FUNCTION_BLOCK FB_LA
VAR_INPUT

	Modbus_LA		: BOOL;
END_VAR
VAR_IN_OUT
END_VAR
VAR_OUTPUT
END_VAR
VAR
(*Diagnose-Funktion stellt eine Reihe von Tests für die Überprüfung des Übertragungssystems zwischen dem Master und dem Slave,
oder für die Überprüfung der verschiedenen internen Fehlerzustände innerhalb des Slaves, zur Verfügung.*)
	LA_955_Diagnose	: FB_MBDiagnose;
	IPAddr	 		: STRING(15);(* IPv4 address of the target device *)
	TCPPort			: UINT:= MODBUS_TCP_PORT;(* Port number of the target device *)
	UnitID			: BYTE:=16#FF;(* Identification number of a serial sub-network device *)
	WriteData		: WORD;
	Execute			: BOOL;(* Rising edge at this input starts command execution *)
	Timeout			: TIME;
	SubFnc			: WORD;
	Diagnose		: BOOL;
	Diagnose_busy	: BOOL;
	Diagnose_Error	: BOOL;
	Diagnose_ErrorID: UDINT;
	Read_Data		: WORD;

(* FB_MBReadRegs*)
	(* Read 1..128 input registers (word access) *)
	LA_955_ReadRegs		: FB_MBReadRegs;
	DestAddrRR			: PVOID;(* Pointer to destination buffer *)
	LA955_RR_arrData	: ARRAY [1..26] OF INT;
	ReadRegsBusy_Modus	: BOOL;
	ReadRegsError_Modus	: BOOL;
	ReadRegsErrID_Modus	: UDINT;
	ReadRegsCount_Modus	: UDINT;

(* FB_MBReadInputs *)
	LA_955_ReadInputs		: FB_MBReadInputs;
	ReadInputsBusy_Modus	: BOOL;
	ReadInputs_Error_Modus	: BOOL;
	ReadInputsErrID_Modus	: UDINT;
	ReadInputsCount_Modus	: UDINT;
	LA955_RI_arrData		: ARRAY [1..31] OF BYTE;
	DestAddrInputs			: PVOID;(* Pointer to destination buffer *)

(* FB_MBWriteRegs *)
	LA_955_WriteRegs		: FB_MBWriteRegs;
	WriteRegsBusy_Modus		: BOOL;
	WriteRegs_Error_Modus	: BOOL;
	WriteRegsErrID_Modus	: UDINT;
    LA955_WR_arrData		: ARRAY [1..43] OF INT;
	SrcAddrWR				: PVOID;(* Pointer to source buffer *)

(* FB_MBWritecoils / Coils = einzelner Ein-/ausgang *)
	LA_955_WriteCoils		: FB_MBWriteCoils;
	WriteCoilsBusy_Modus	: BOOL;
	WriteCoils_Error_Modus	: BOOL;
	WriteCoilsErrID_Modus	: UDINT;
    LA955_WC_arrData		: ARRAY [1..42] OF BYTE;
	SrcAddrWC				: PVOID;(* Pointer to source buffer *)

	Aktivieren5			: BOOL;
	Aktivieren6			: BOOL;
	Ablufttemp			: REAL;

(* Blinker *)
	Blinker_Abfrage		: BOOL;
	T_on				: TIME:=t#2s;
	T_off				: TIME:=t#1s;
	Timer1				: TON;
	Timer2				: TON;

	{attribute 'OPC.UA.DA' := '1'}Steuerung		: ST_LA_Steuerung; 
	{attribute 'OPC.UA.DA' := '1'}Parameter		: ST_LA_Parameter; 
	{attribute 'OPC.UA.DA' := '1'}Stellwert		: ST_LA_Stellwert; 
	{attribute 'OPC.UA.DA' := '1'}Zustand			: ST_LA_Zustand;
	Zustandscheck	: FB_LA_Zustandscheck;
END_VAR
VAR // added by the converter: edge detectors and wires of the graphical bodies
    _w1, _w2, _w3, _w4, _w5, _w6, _w7, _w8, _w9, _w10, _w11, _w12, _w13, _w14, _w15, _w16, _w17, _w18, _w19, _w20, _w21, _w22, _w23, _w24, _w25, _w26, _w27, _w28, _w29, _w30, _w31, _w32 : ANY;
END_VAR

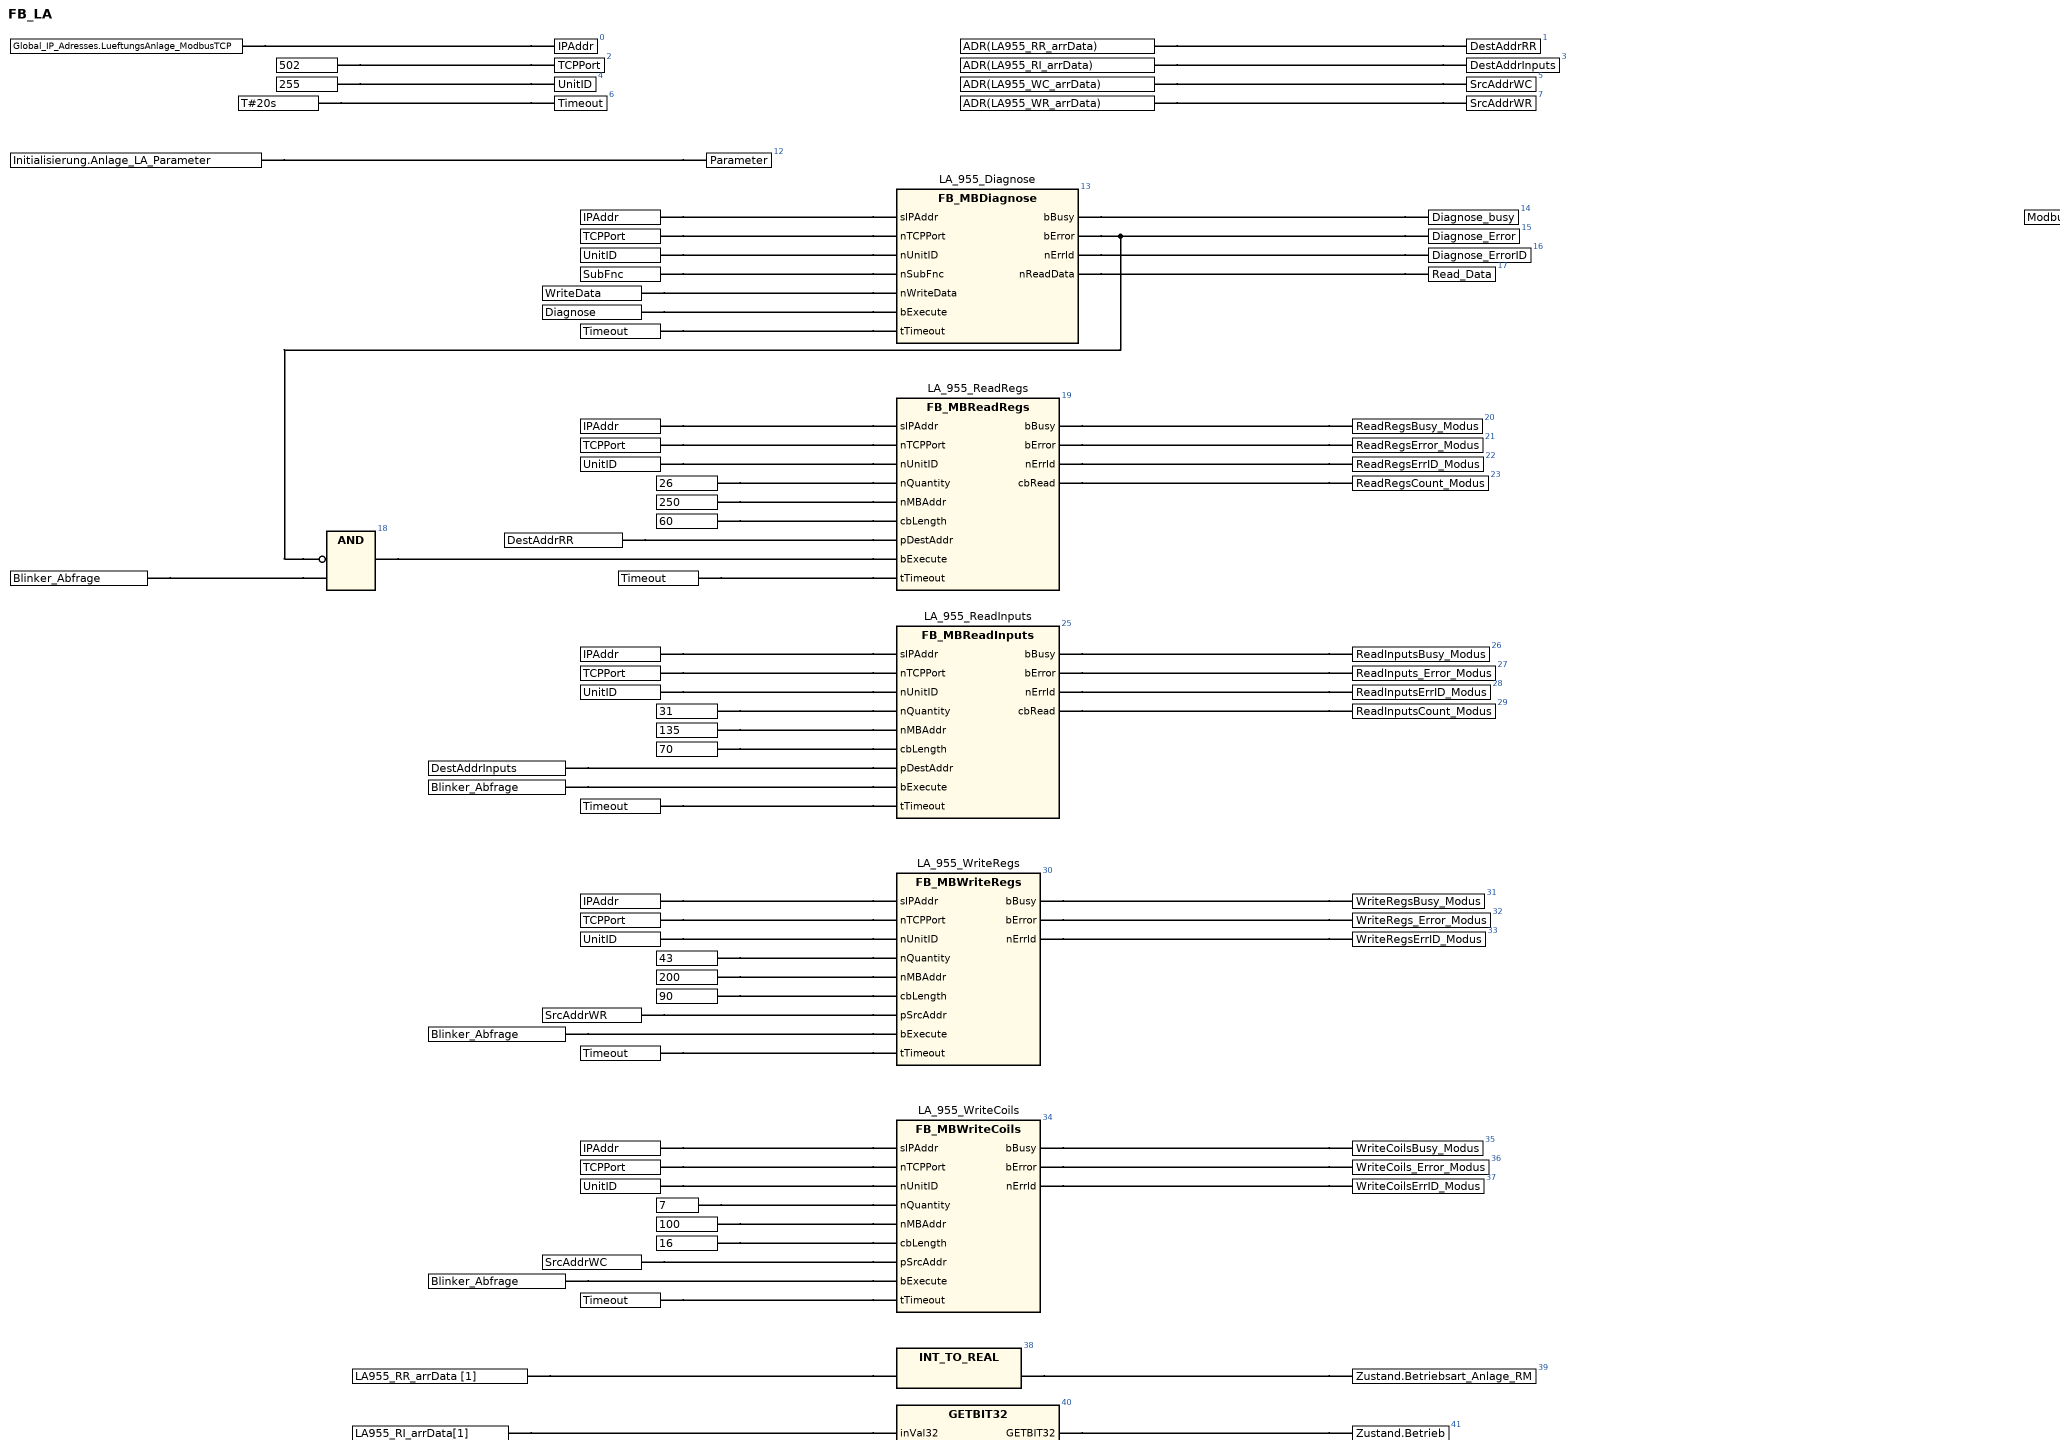
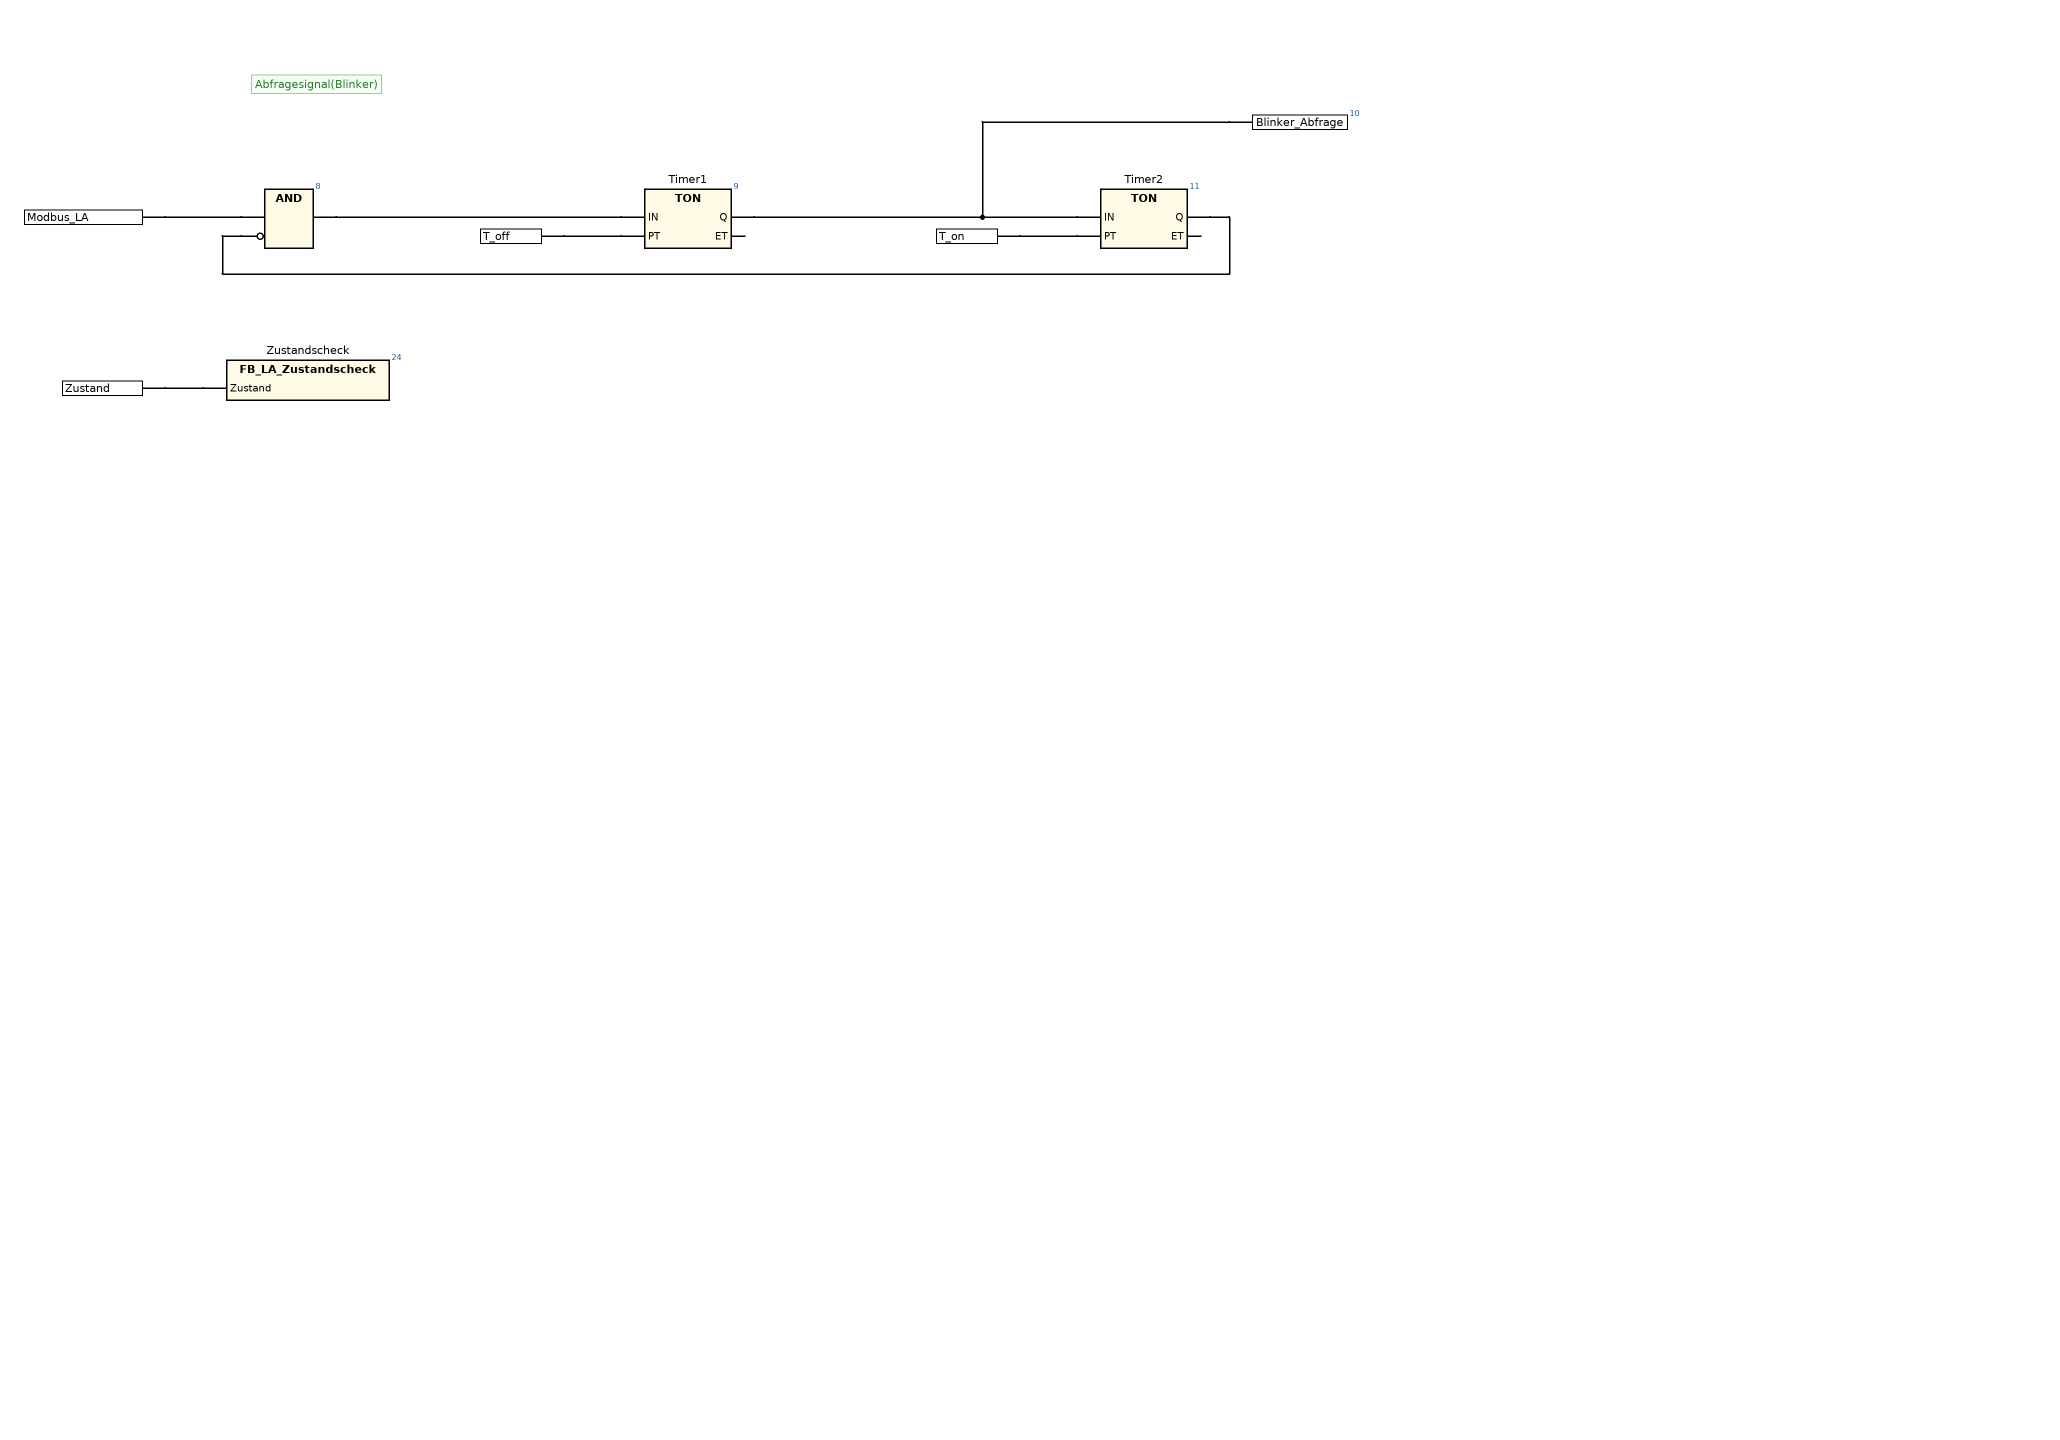
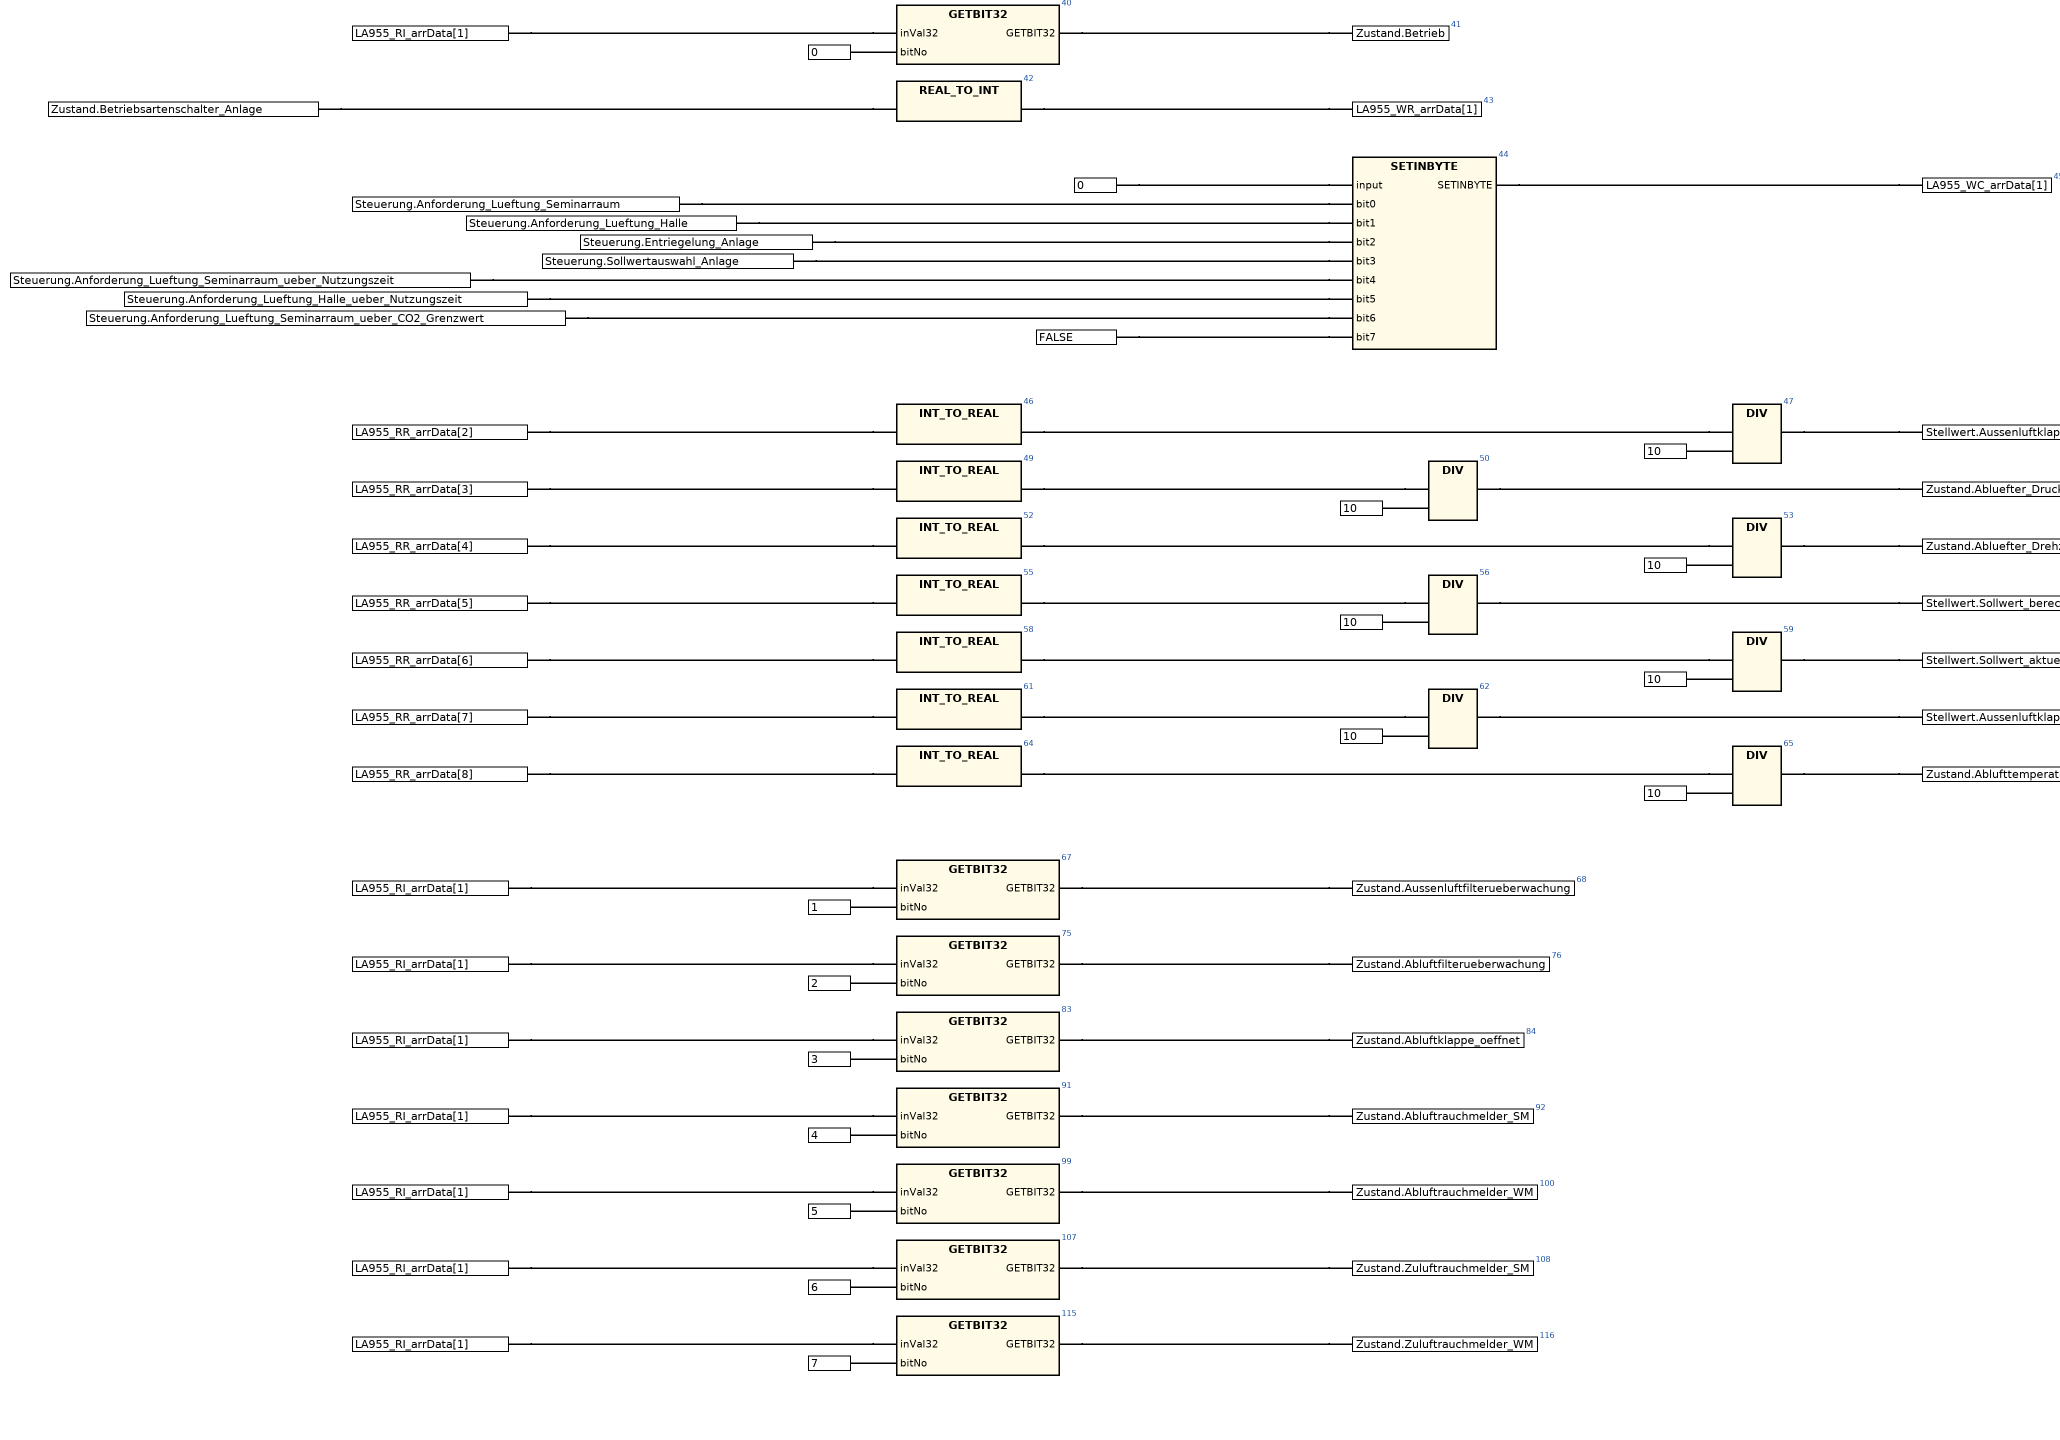
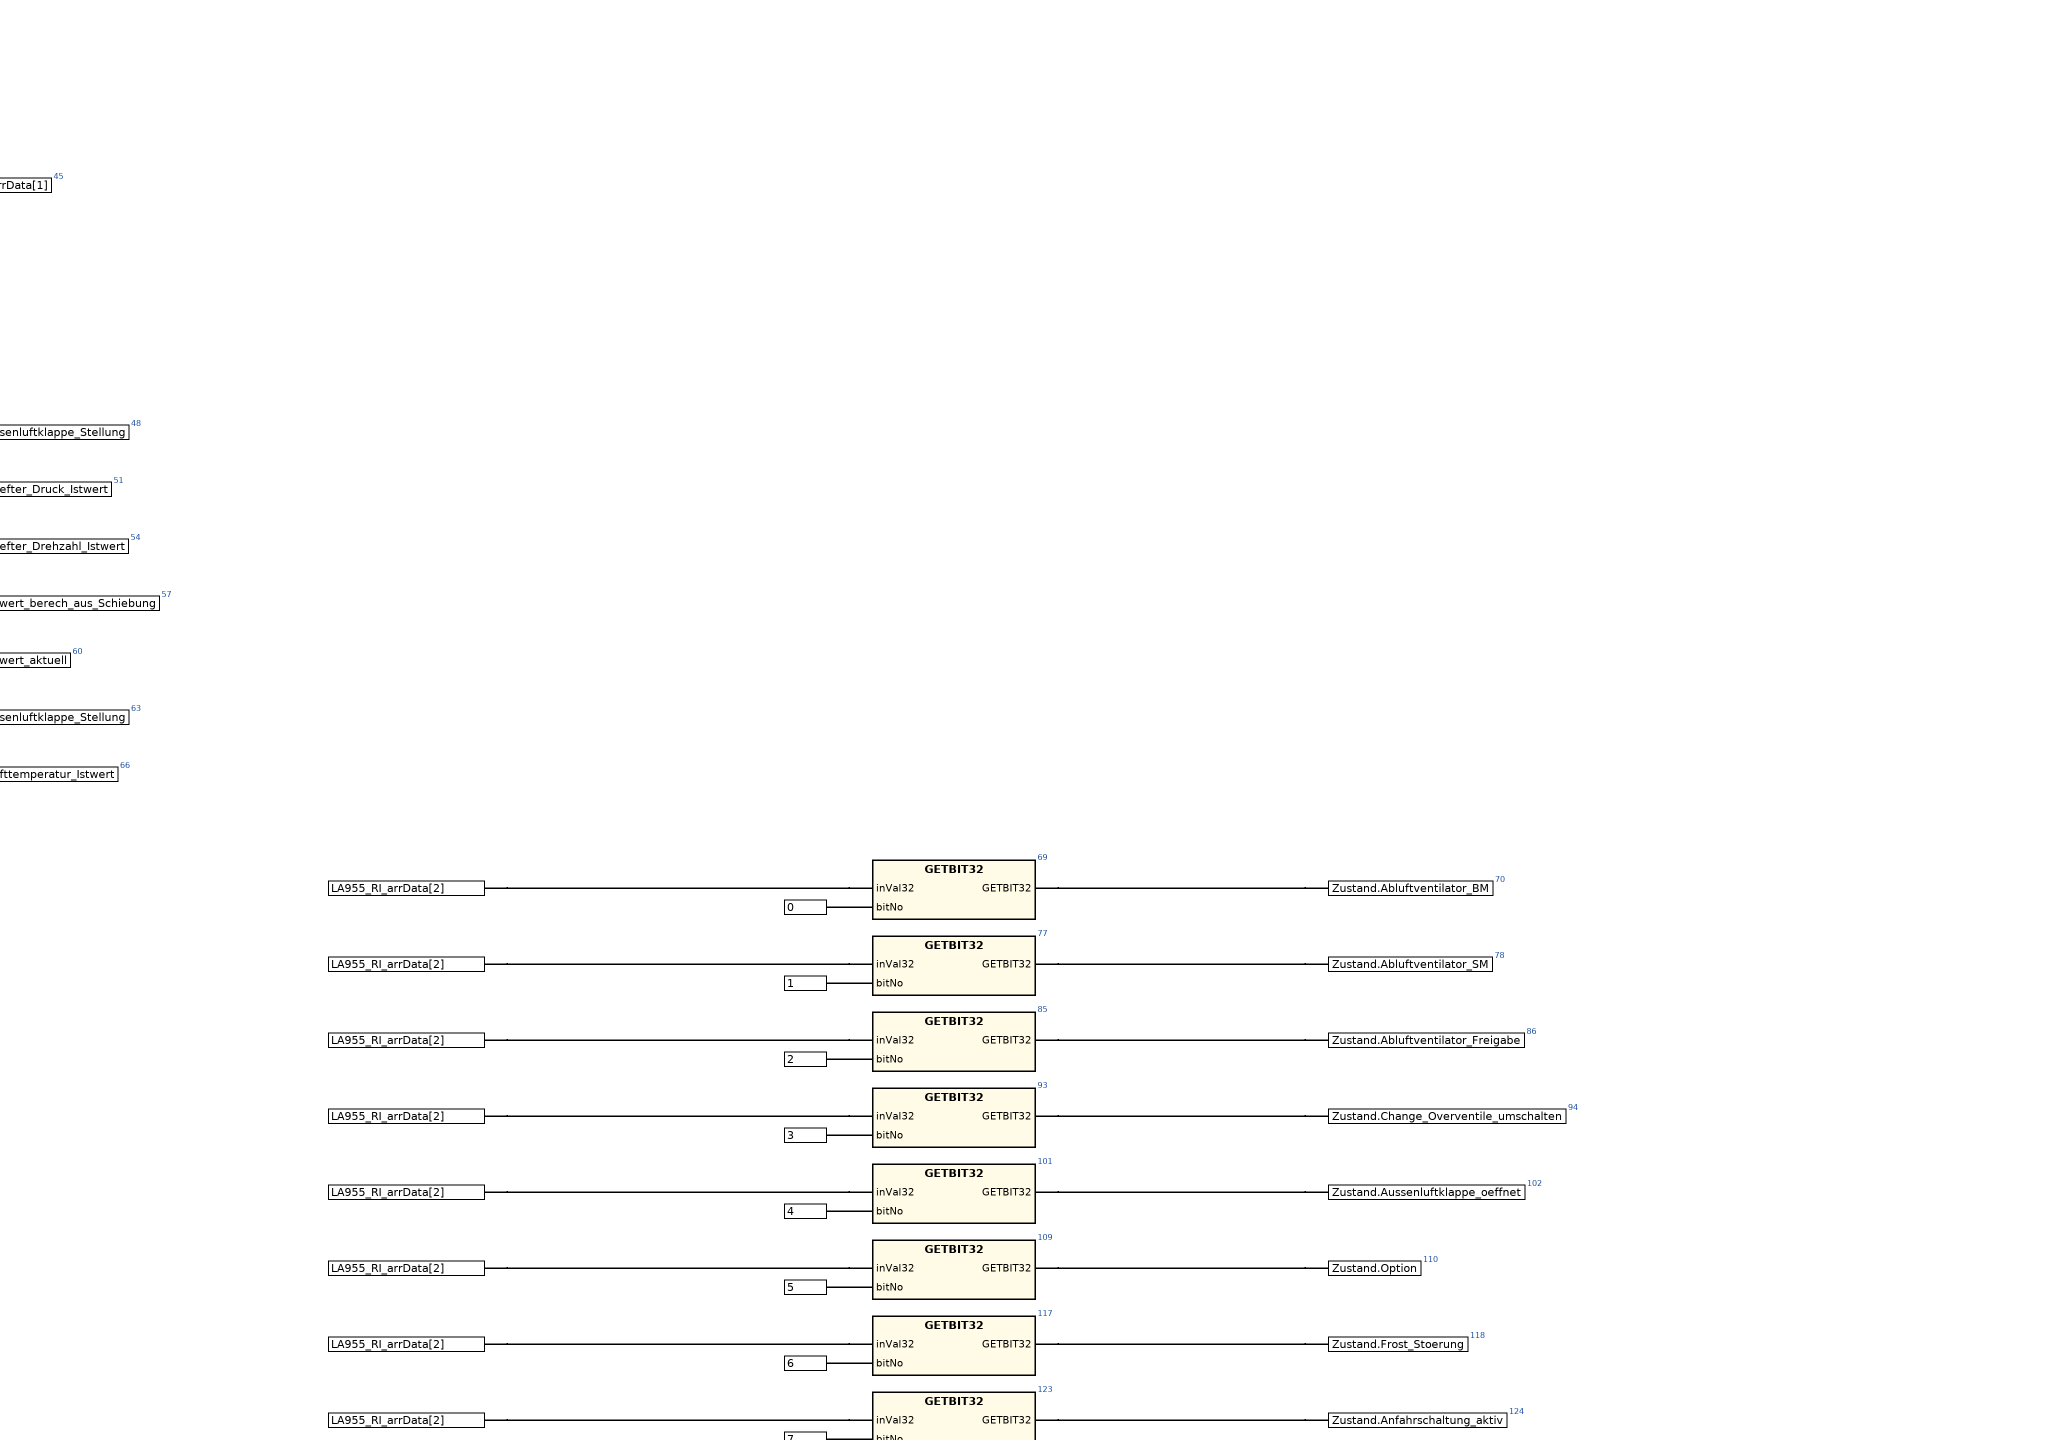
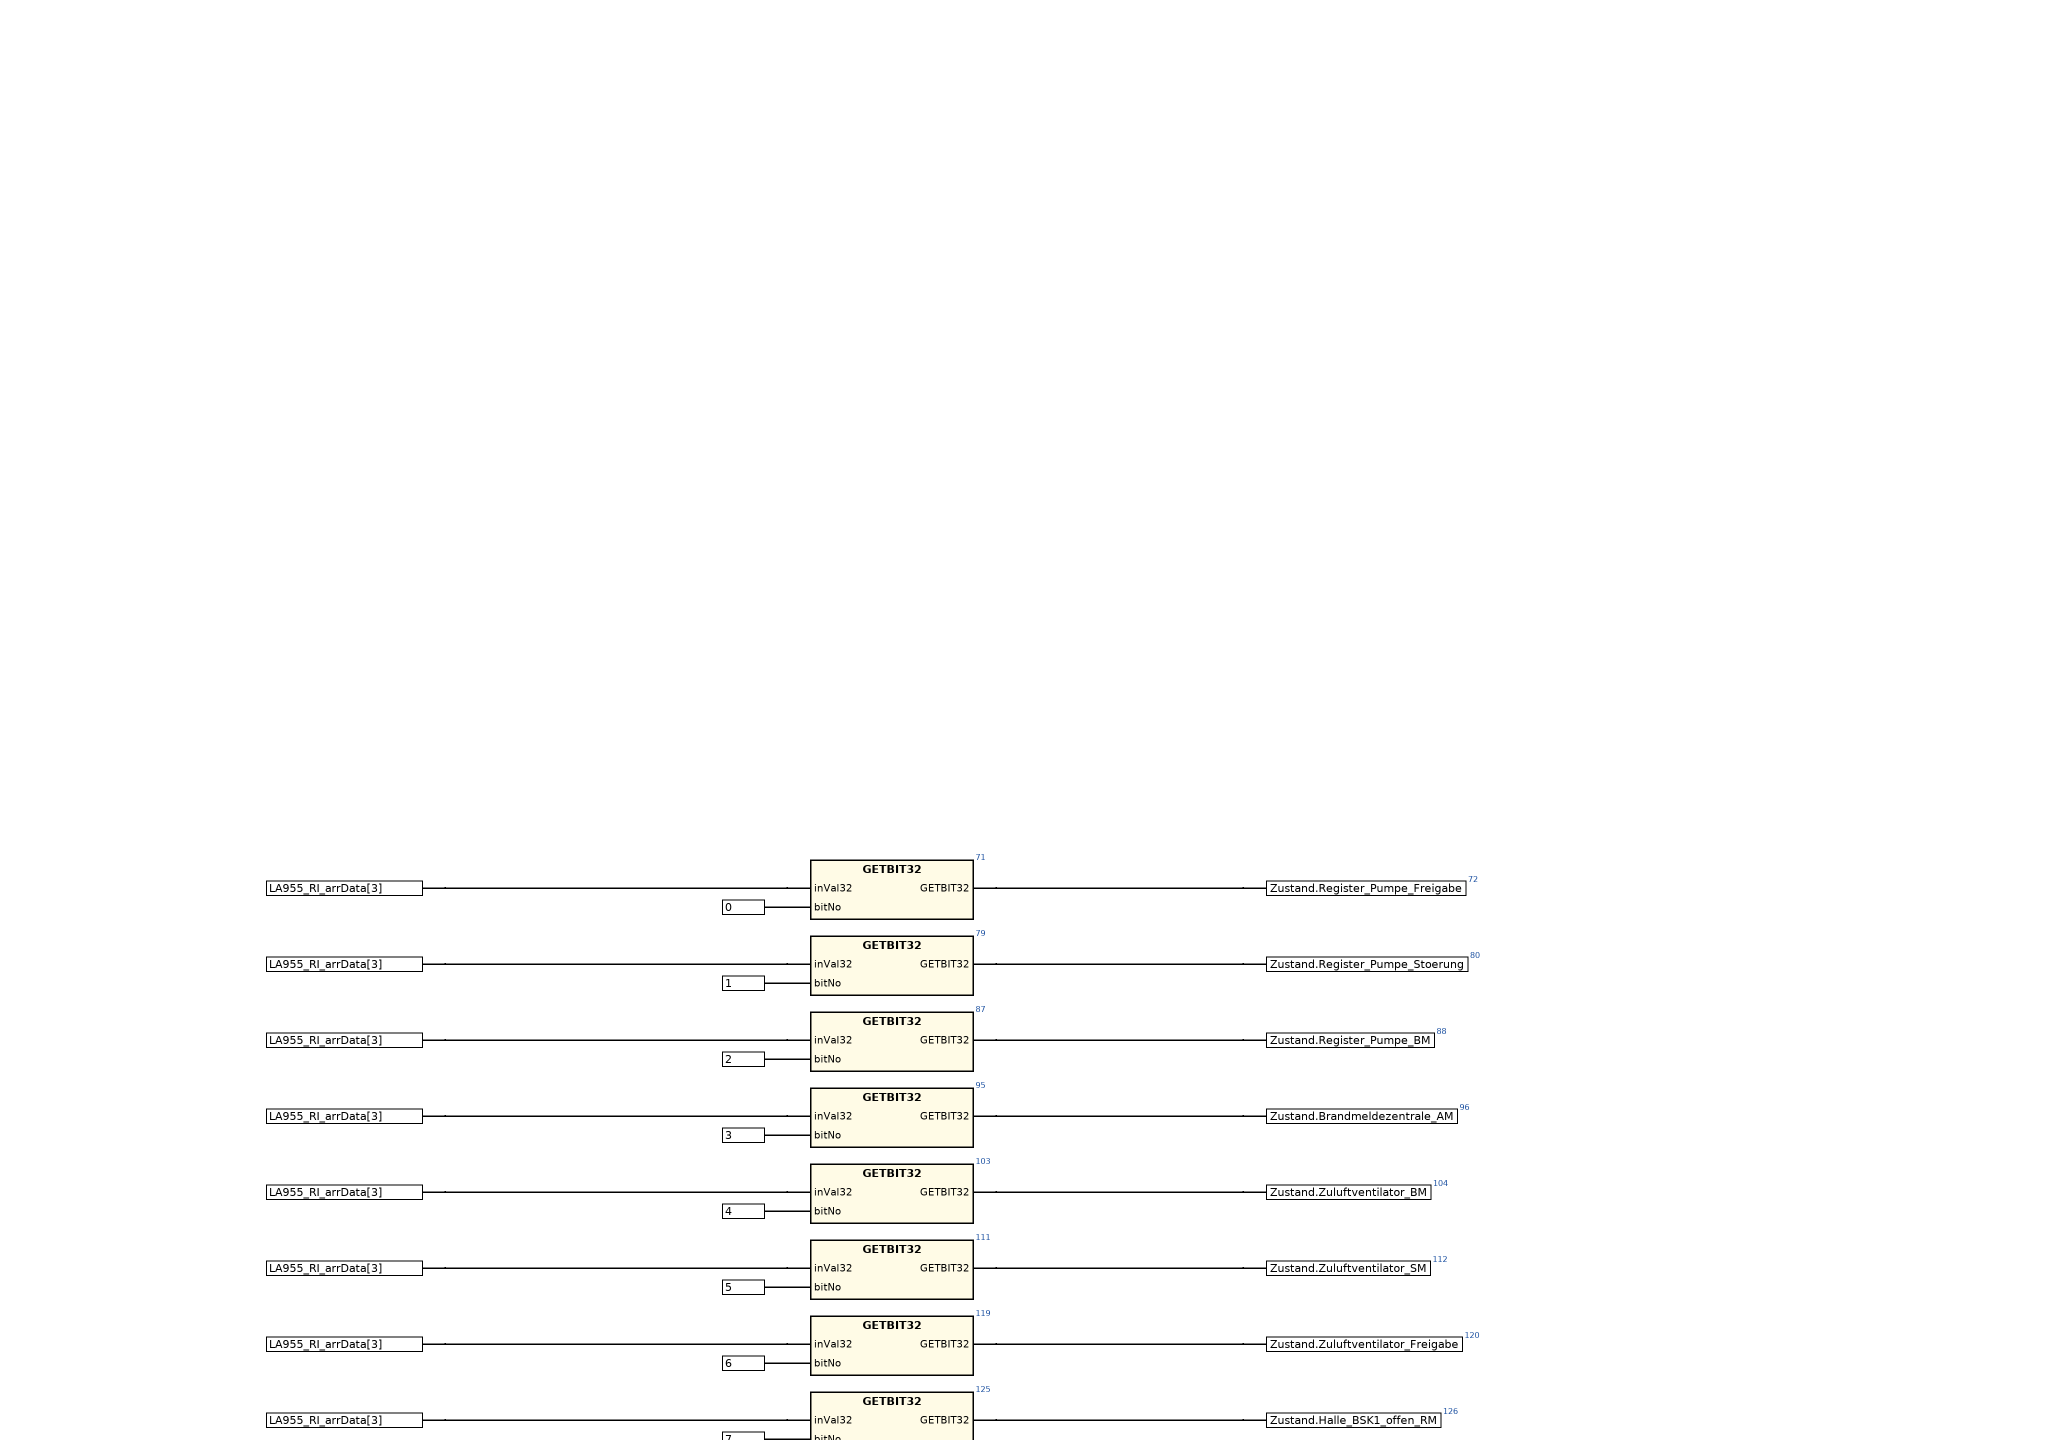
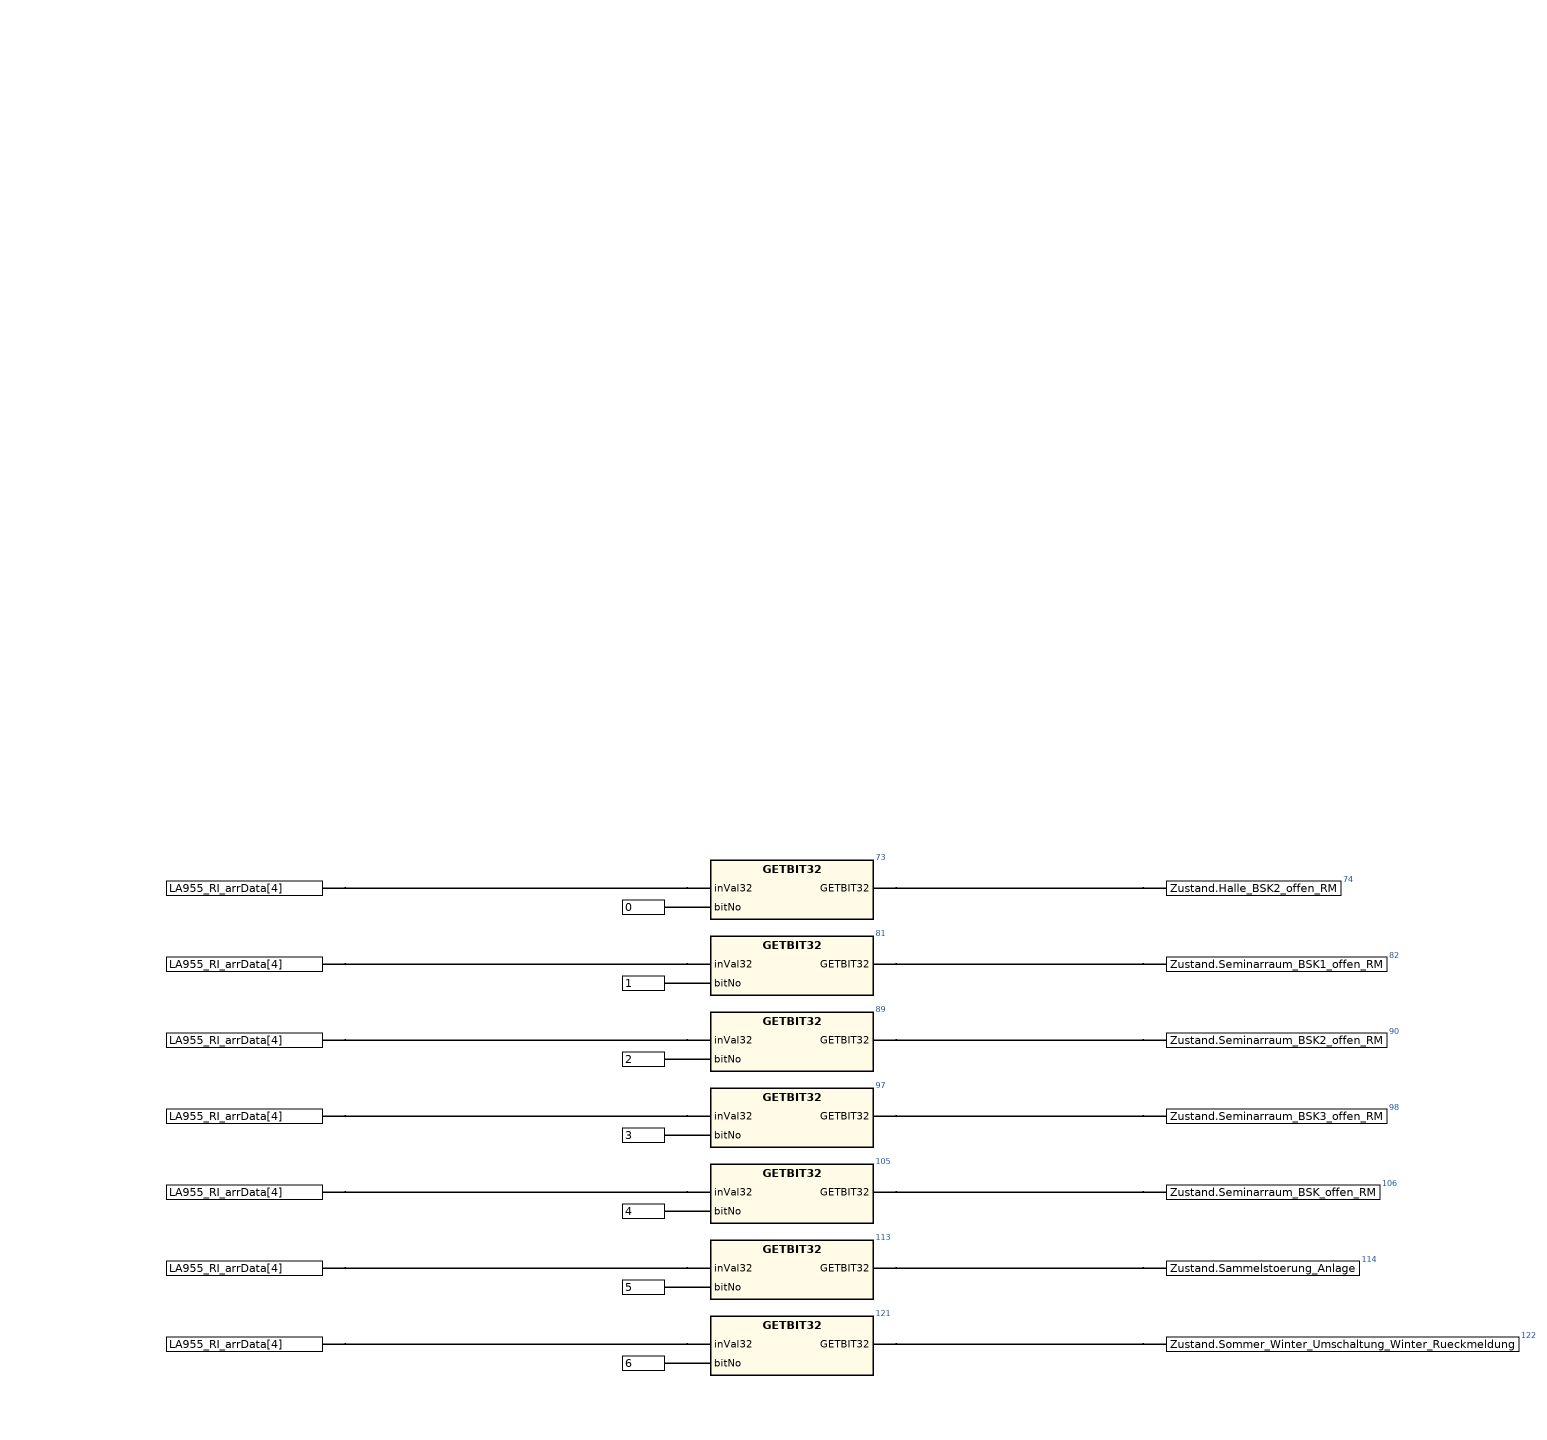
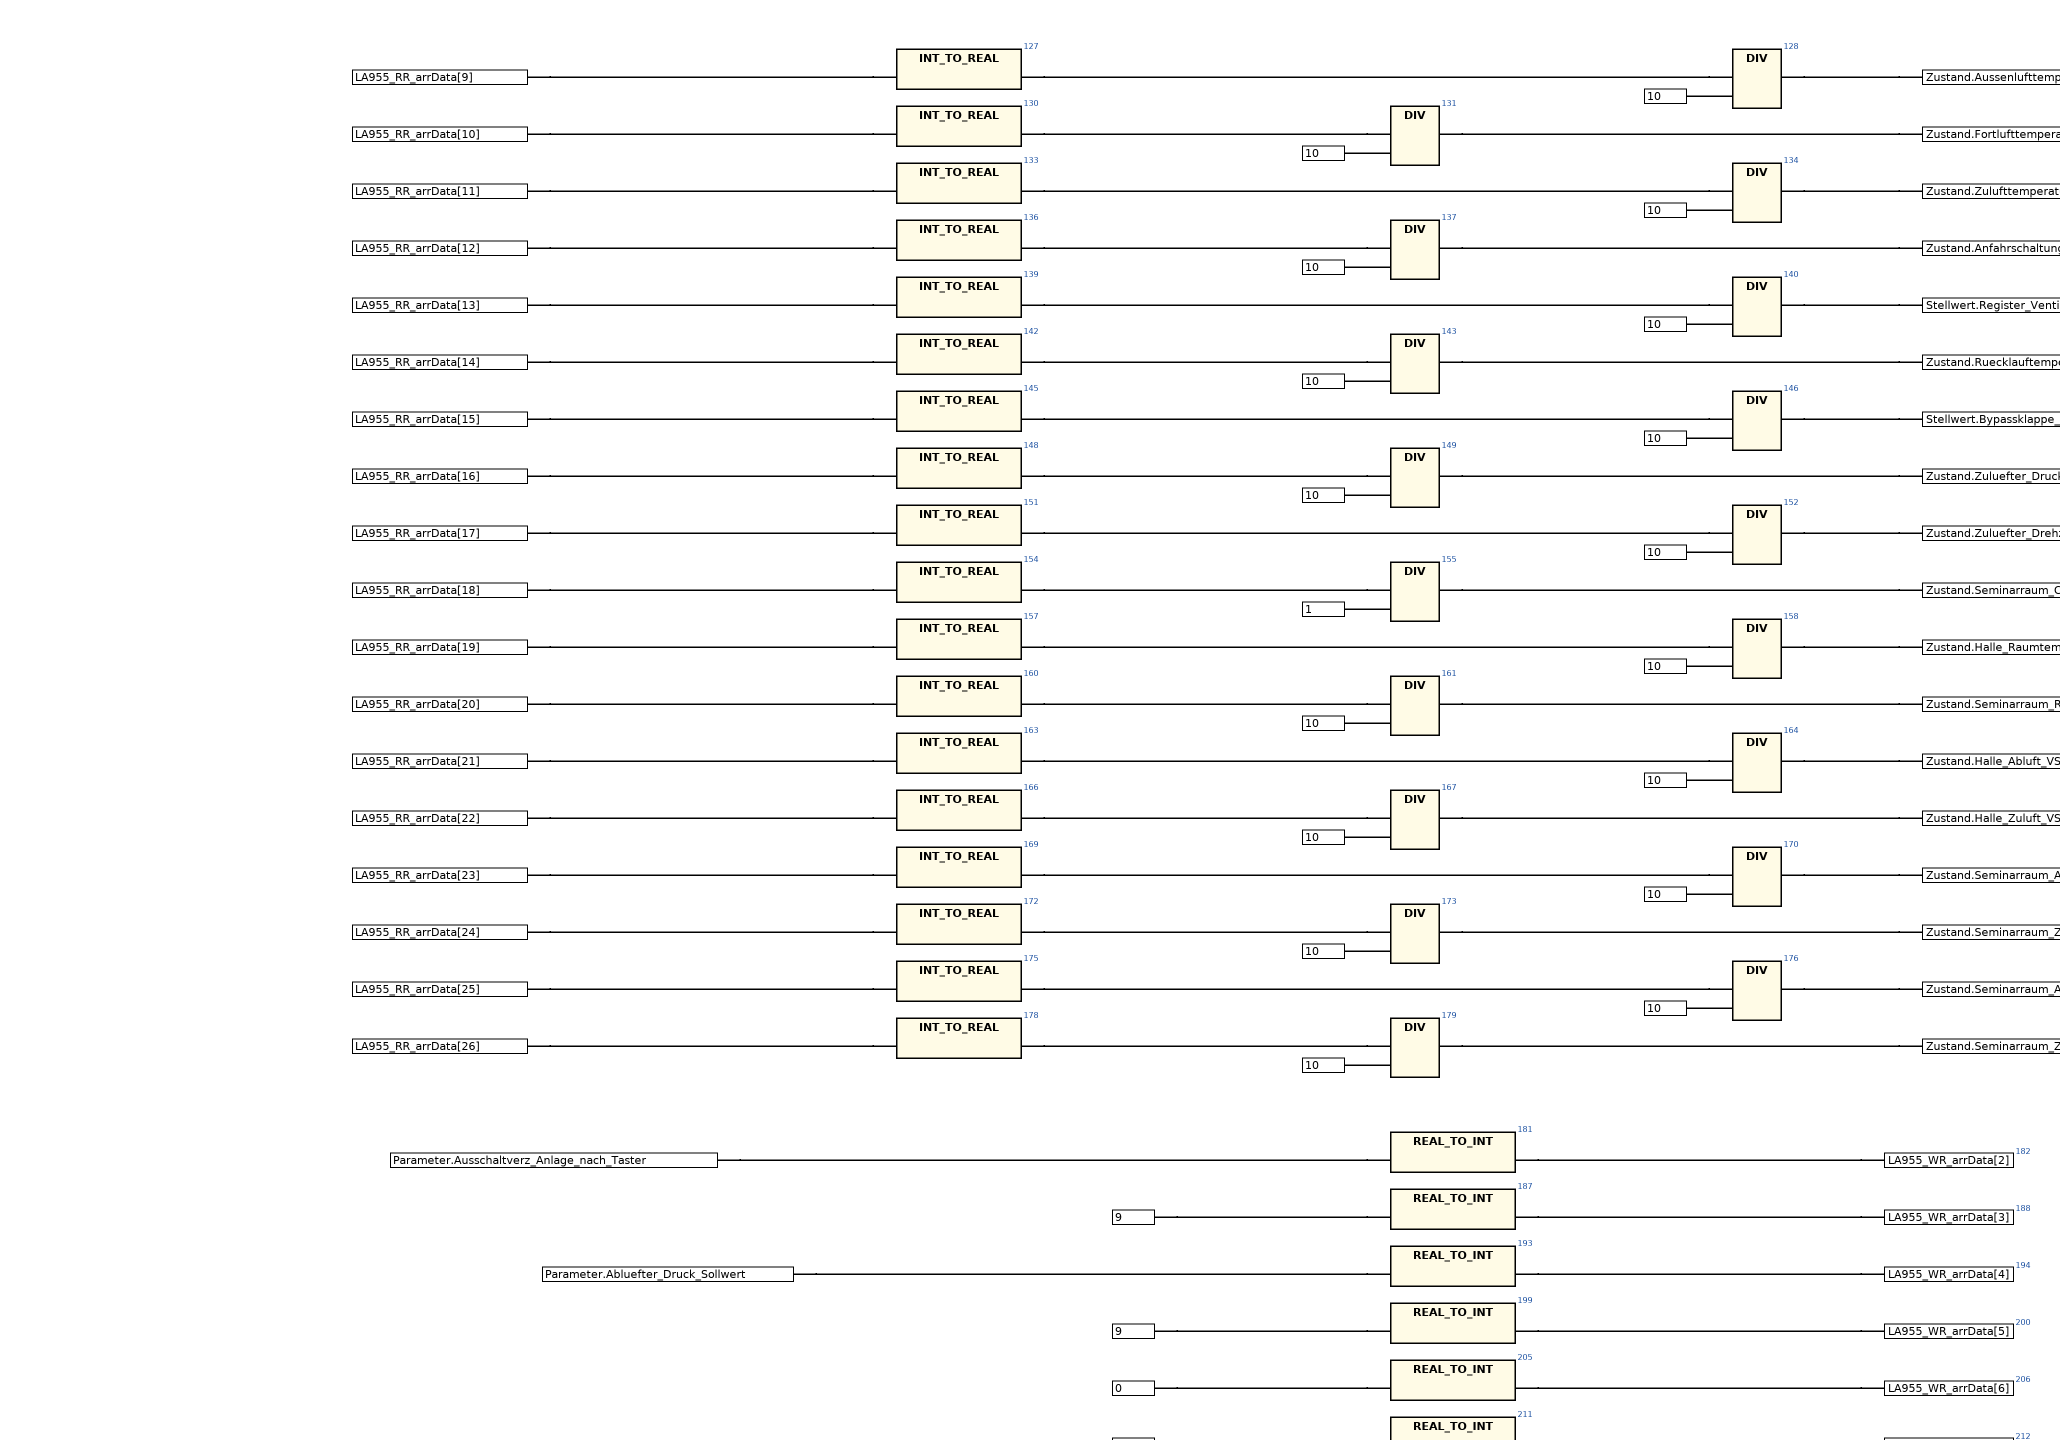
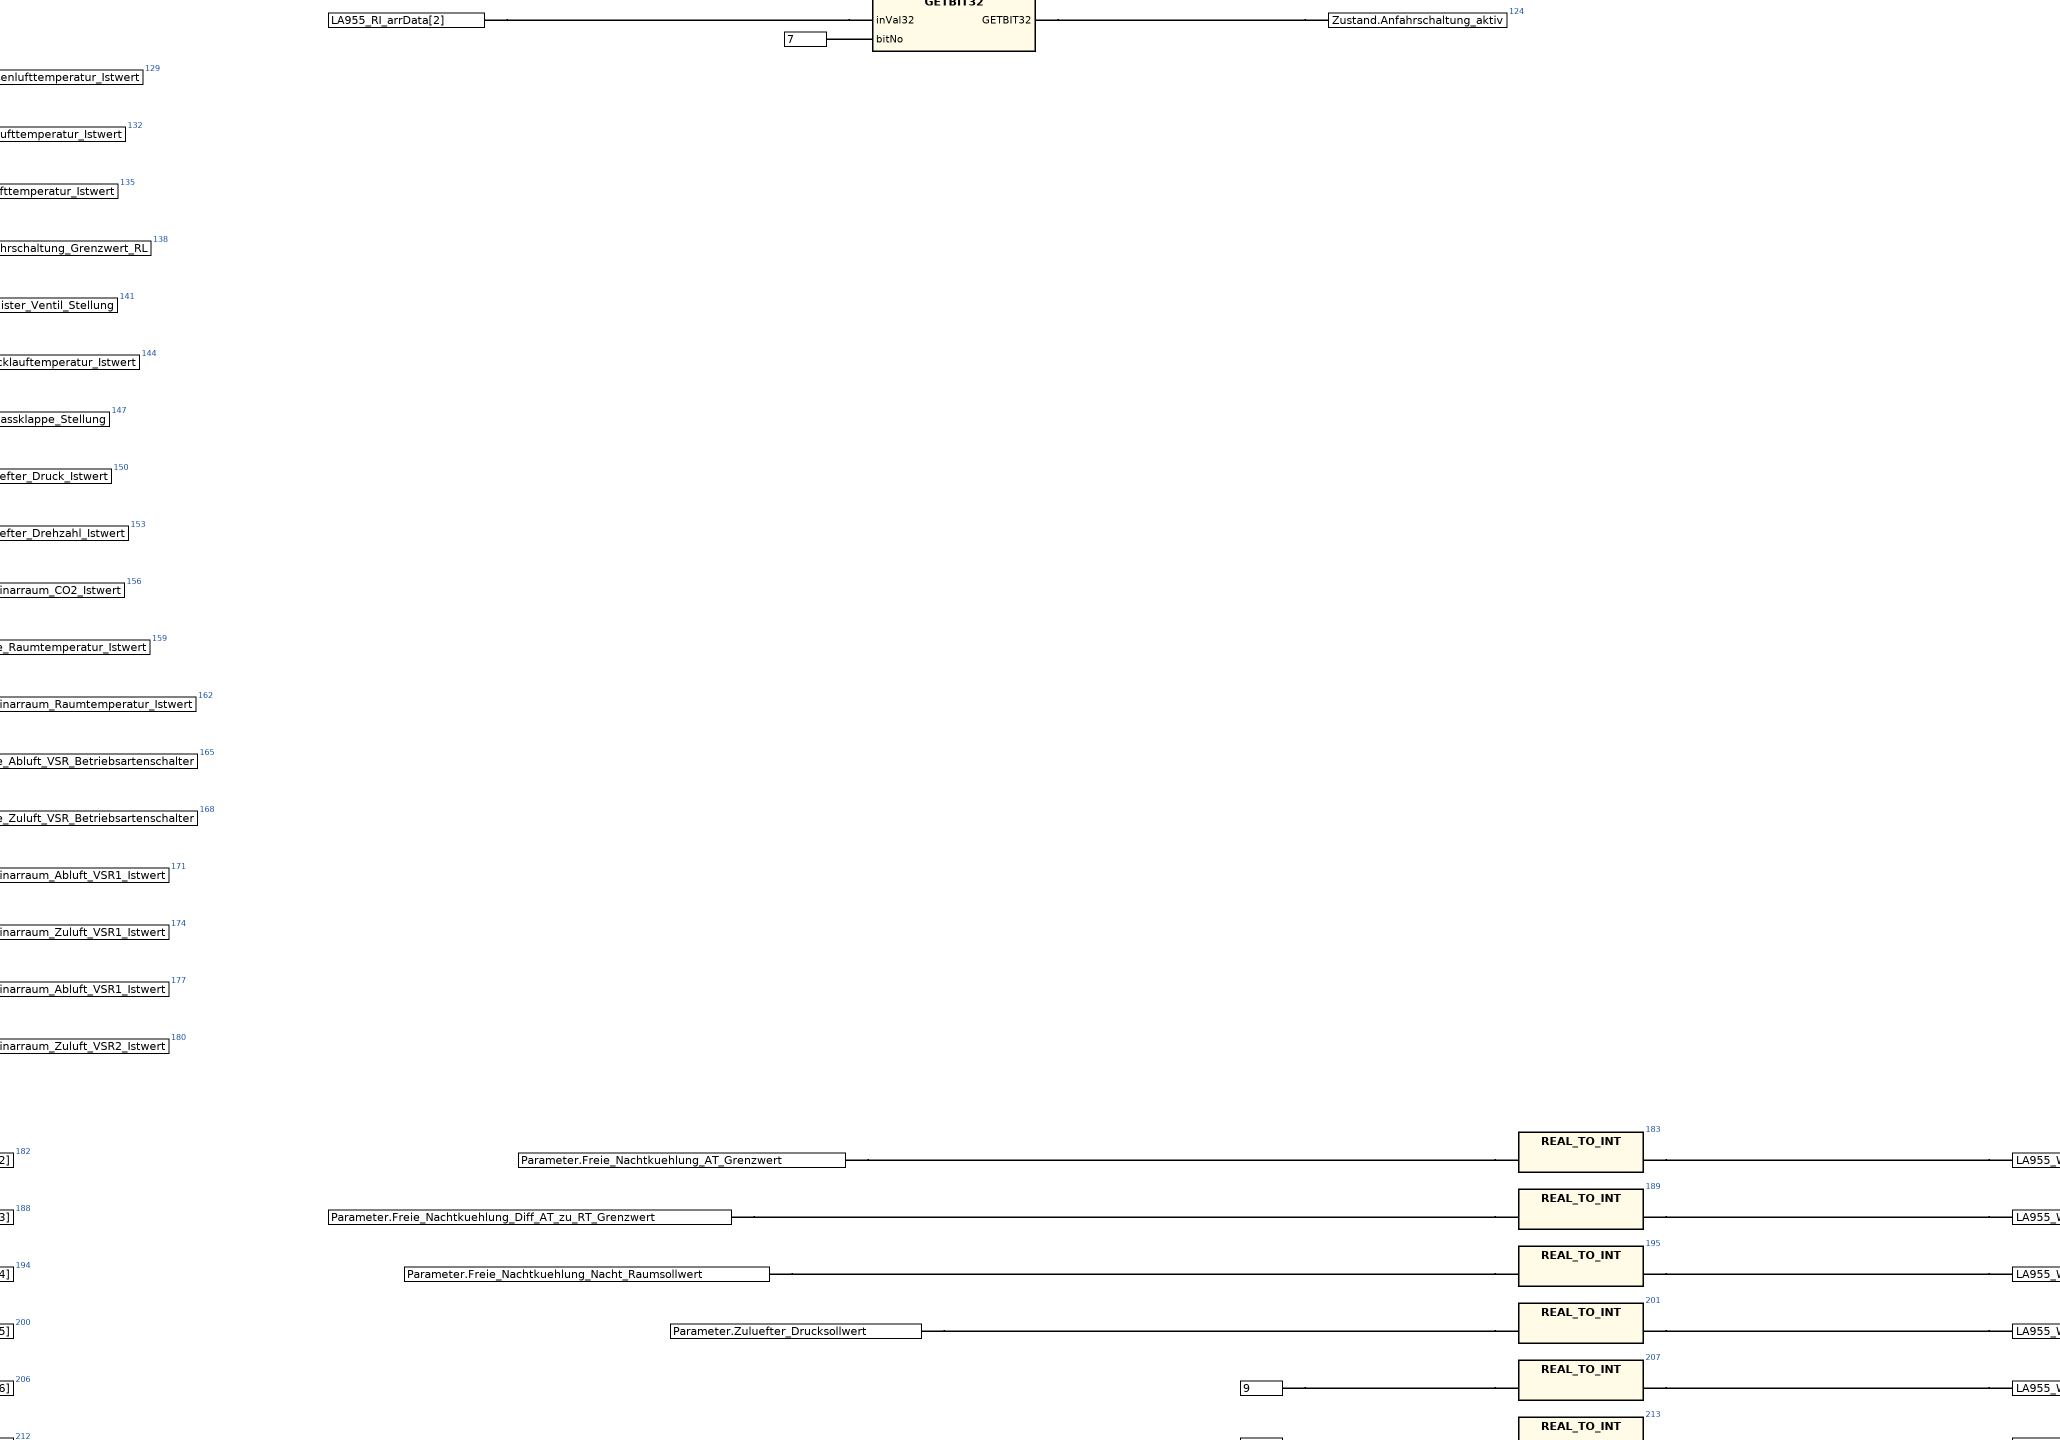
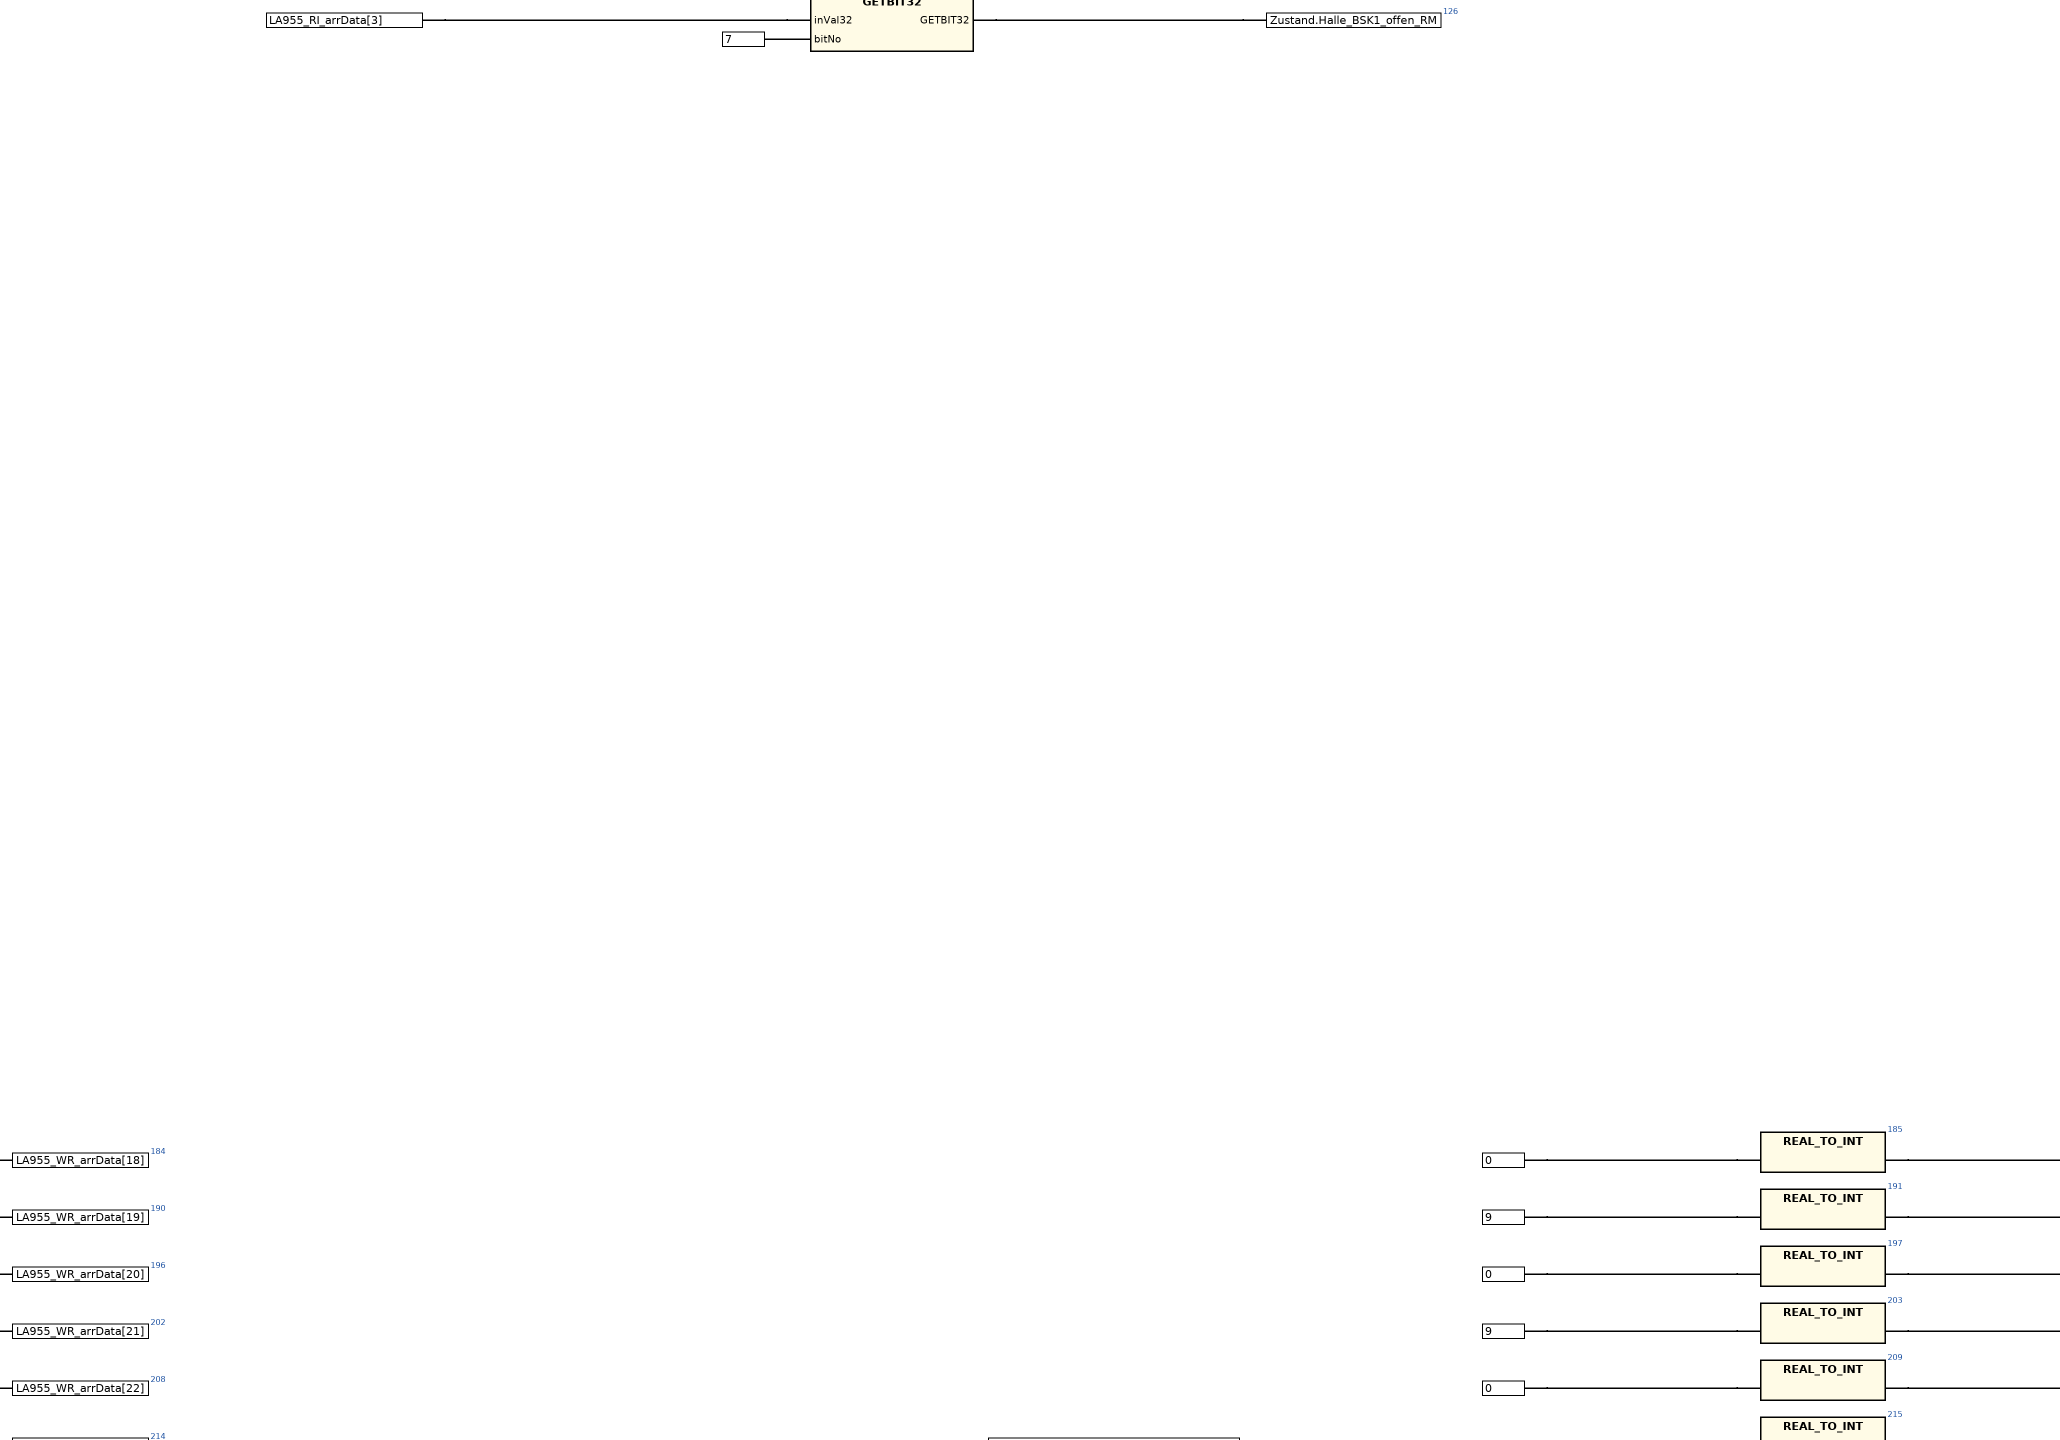
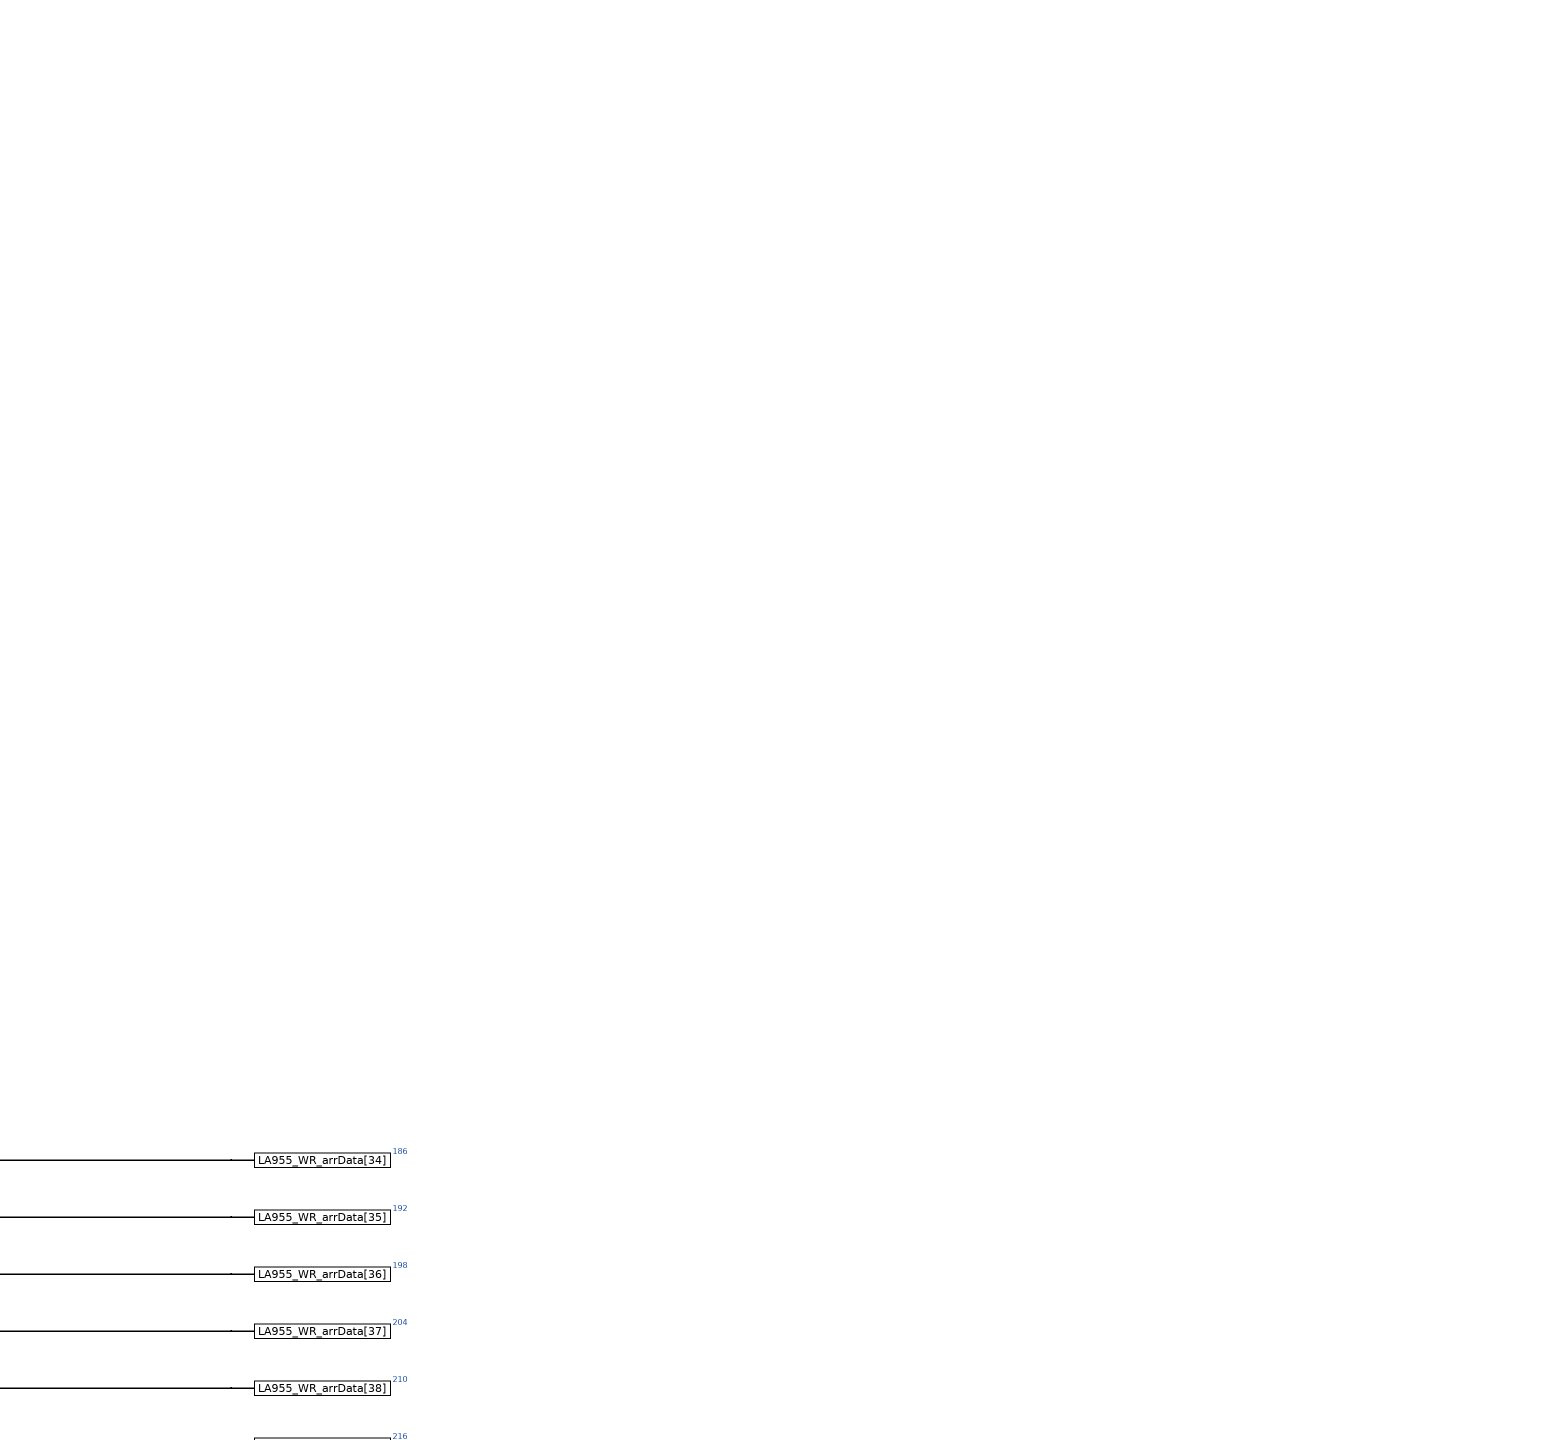
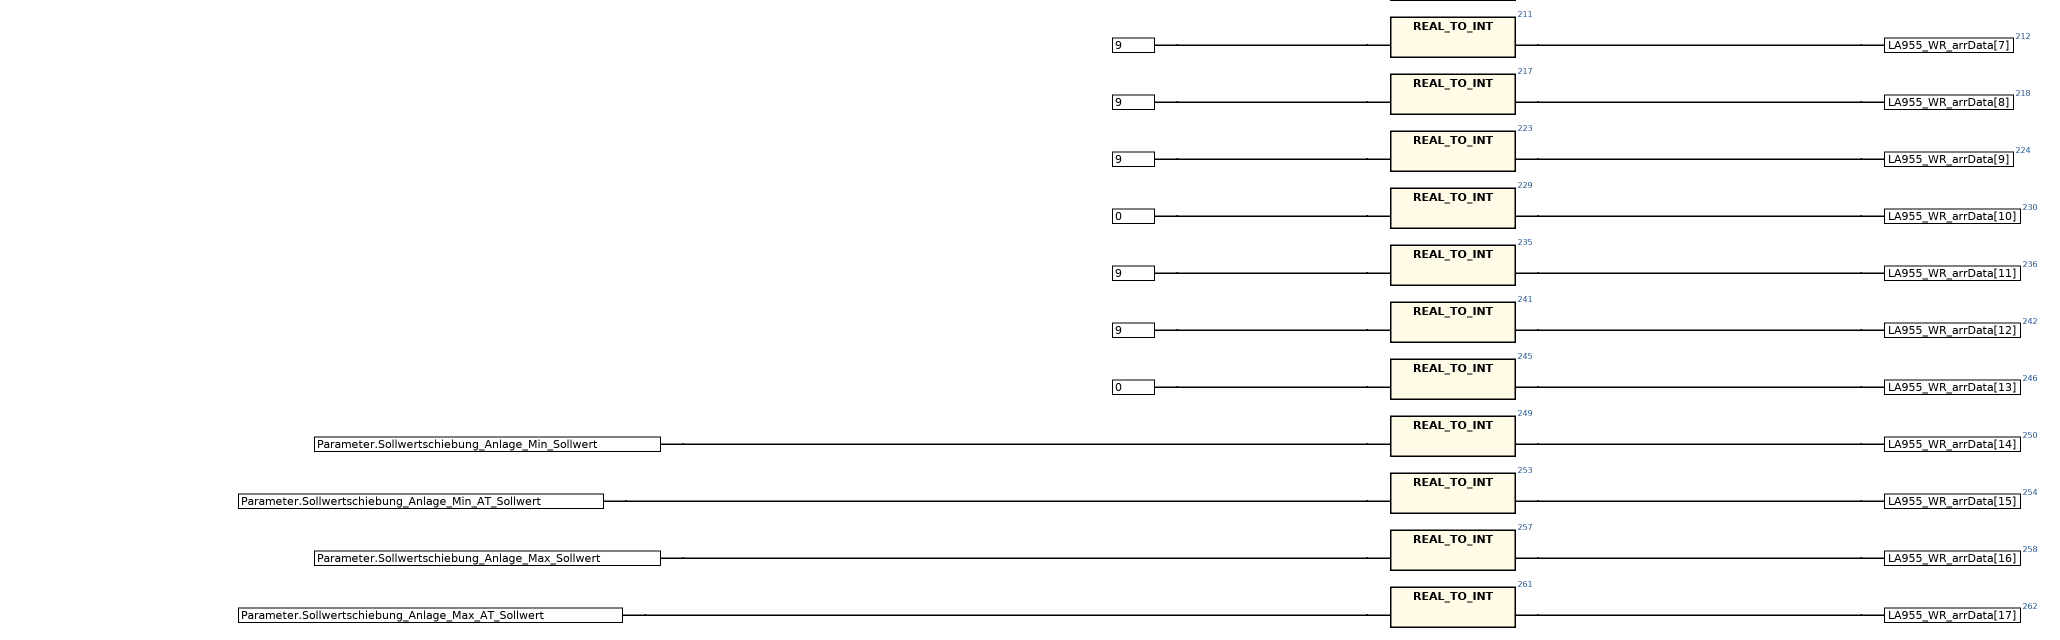
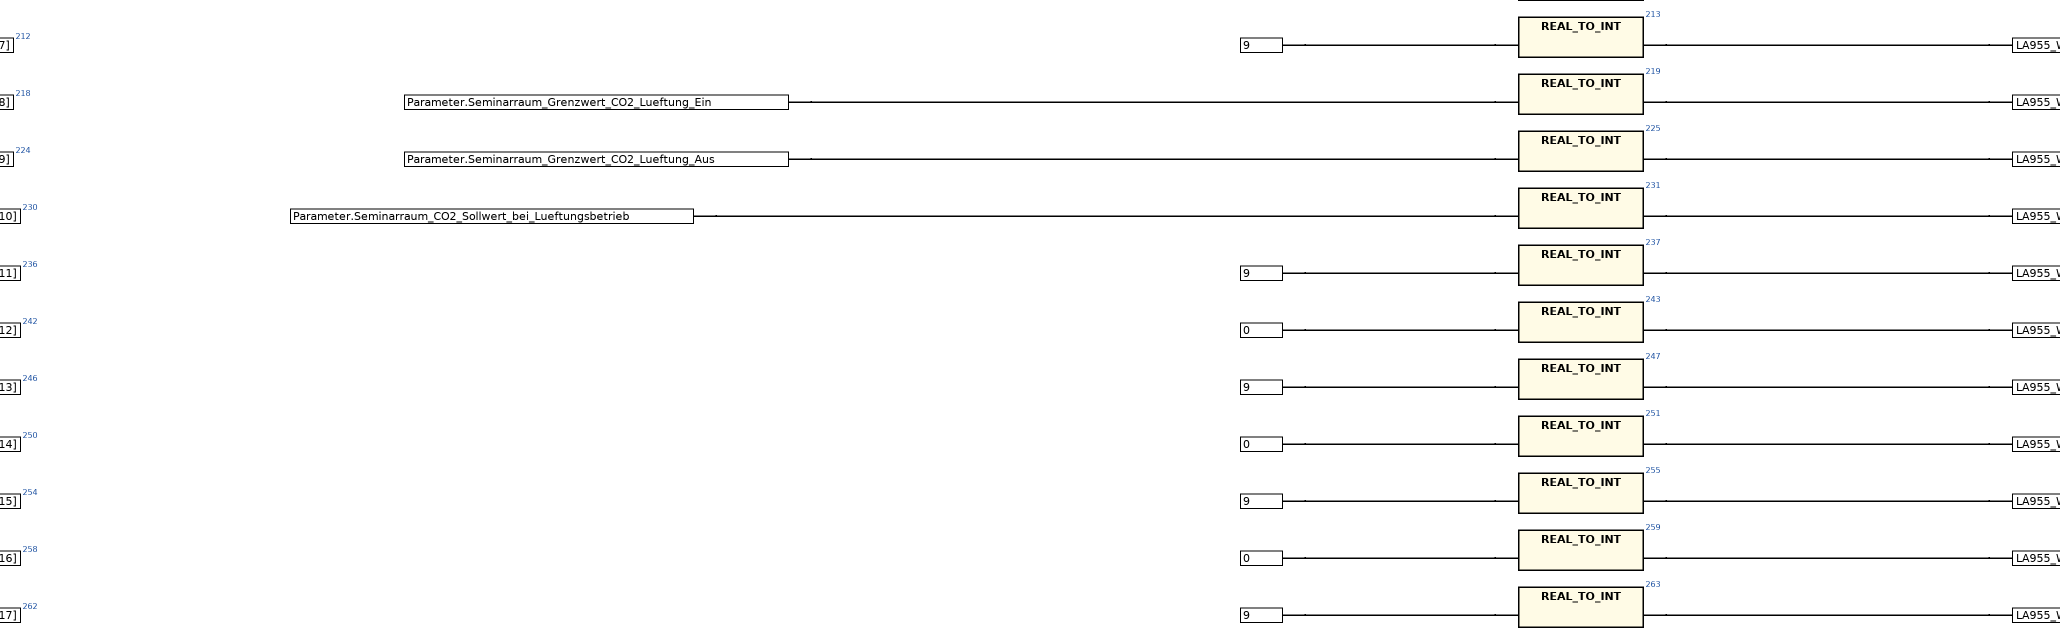
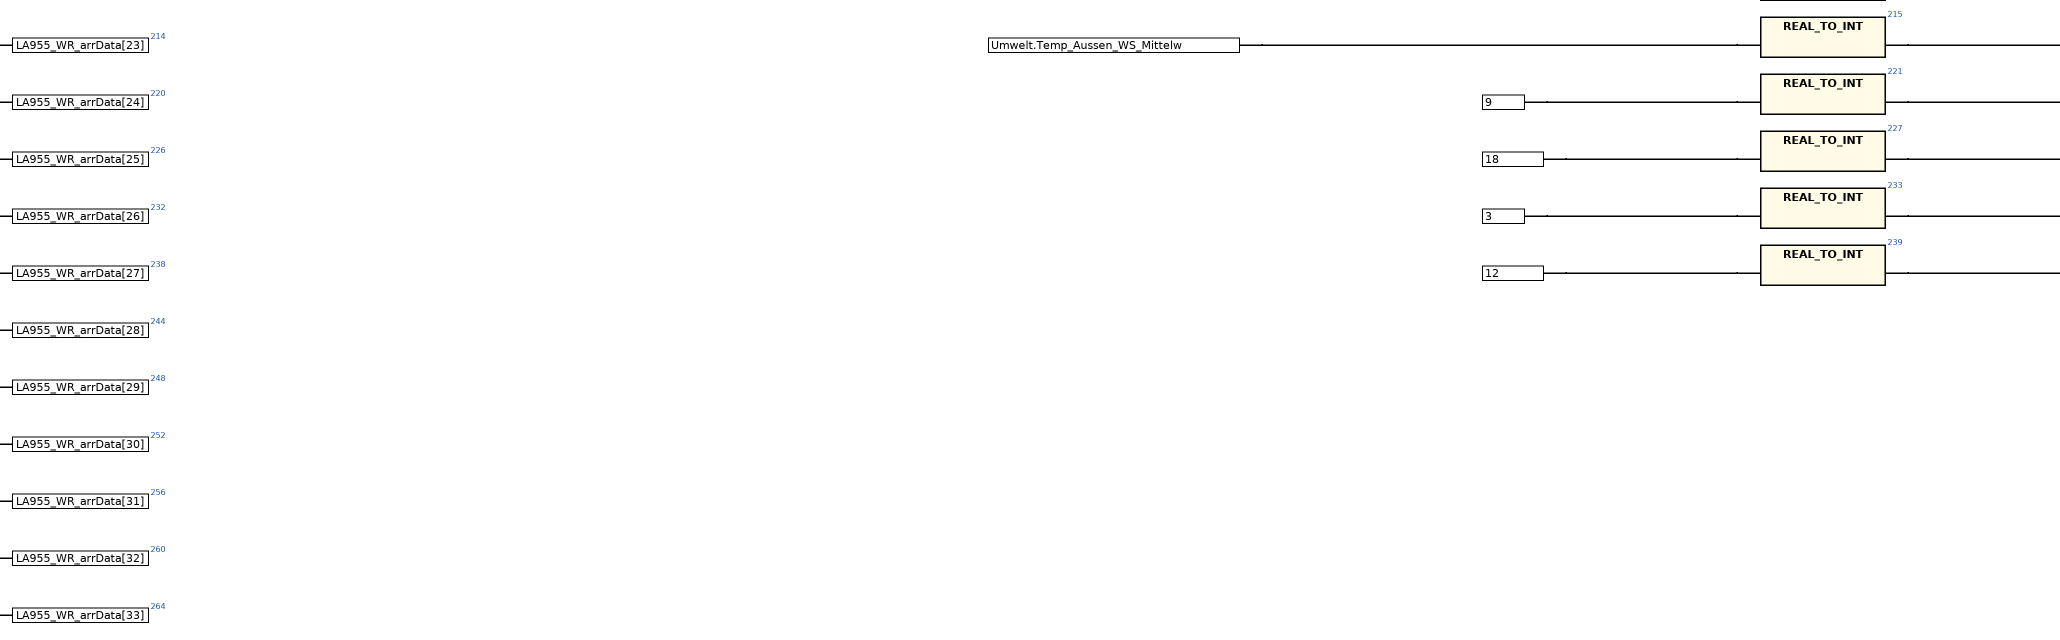
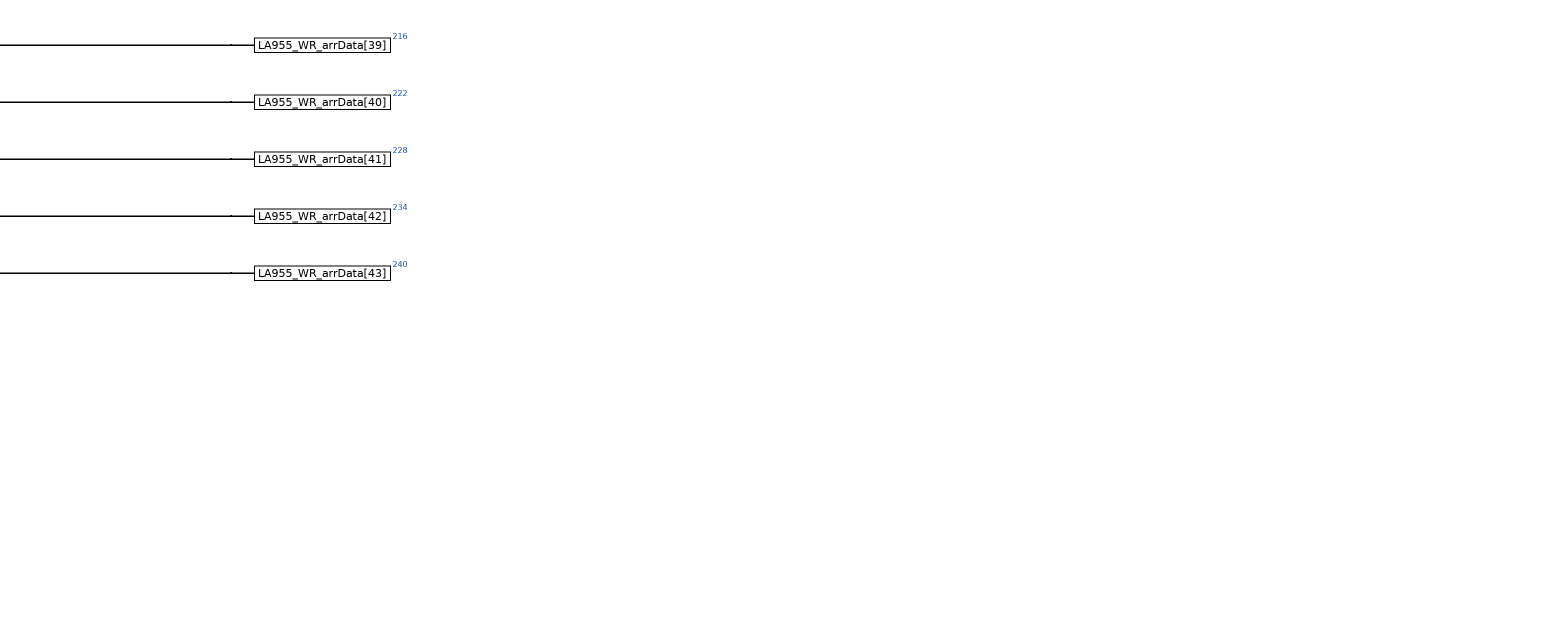
IPAddr := Global_IP_Adresses.LueftungsAnlage_ModbusTCP;
DestAddrRR := ADR(LA955_RR_arrData);
TCPPort := 502;
DestAddrInputs := ADR(LA955_RI_arrData);
UnitID := 255;
SrcAddrWC := ADR(LA955_WC_arrData);
Timeout := T#20s;
SrcAddrWR := ADR(LA955_WR_arrData);
// Abfragesignal(Blinker)
Timer1(IN := Modbus_LA AND NOT Timer2.Q, PT := T_off); // TON
Blinker_Abfrage := Timer1.Q;
Timer2(IN := Timer1.Q, PT := T_on); // TON
Parameter := Initialisierung.Anlage_LA_Parameter;
LA_955_Diagnose(
    sIPAddr := IPAddr,
    nTCPPort := TCPPort,
    nUnitID := UnitID,
    nSubFnc := SubFnc,
    nWriteData := WriteData,
    bExecute := Diagnose,
    tTimeout := Timeout); // FB_MBDiagnose
Diagnose_busy := LA_955_Diagnose.bBusy;
Diagnose_Error := LA_955_Diagnose.bError;
Diagnose_ErrorID := LA_955_Diagnose.nErrId;
Read_Data := LA_955_Diagnose.nReadData;
LA_955_ReadRegs(
    sIPAddr := IPAddr,
    nTCPPort := TCPPort,
    nUnitID := UnitID,
    nQuantity := 26,
    nMBAddr := 250,
    cbLength := 60,
    pDestAddr := DestAddrRR,
    bExecute := NOT LA_955_Diagnose.bError AND Blinker_Abfrage,
    tTimeout := Timeout); // FB_MBReadRegs
ReadRegsBusy_Modus := LA_955_ReadRegs.bBusy;
ReadRegsError_Modus := LA_955_ReadRegs.bError;
ReadRegsErrID_Modus := LA_955_ReadRegs.nErrId;
ReadRegsCount_Modus := LA_955_ReadRegs.cbRead;
Zustandscheck(Zustand := Zustand); // FB_LA_Zustandscheck
LA_955_ReadInputs(
    sIPAddr := IPAddr,
    nTCPPort := TCPPort,
    nUnitID := UnitID,
    nQuantity := 31,
    nMBAddr := 135,
    cbLength := 70,
    pDestAddr := DestAddrInputs,
    bExecute := Blinker_Abfrage,
    tTimeout := Timeout); // FB_MBReadInputs
ReadInputsBusy_Modus := LA_955_ReadInputs.bBusy;
ReadInputs_Error_Modus := LA_955_ReadInputs.bError;
ReadInputsErrID_Modus := LA_955_ReadInputs.nErrId;
ReadInputsCount_Modus := LA_955_ReadInputs.cbRead;
LA_955_WriteRegs(
    sIPAddr := IPAddr,
    nTCPPort := TCPPort,
    nUnitID := UnitID,
    nQuantity := 43,
    nMBAddr := 200,
    cbLength := 90,
    pSrcAddr := SrcAddrWR,
    bExecute := Blinker_Abfrage,
    tTimeout := Timeout); // FB_MBWriteRegs
WriteRegsBusy_Modus := LA_955_WriteRegs.bBusy;
WriteRegs_Error_Modus := LA_955_WriteRegs.bError;
WriteRegsErrID_Modus := LA_955_WriteRegs.nErrId;
LA_955_WriteCoils(
    sIPAddr := IPAddr,
    nTCPPort := TCPPort,
    nUnitID := UnitID,
    nQuantity := 7,
    nMBAddr := 100,
    cbLength := 16,
    pSrcAddr := SrcAddrWC,
    bExecute := Blinker_Abfrage,
    tTimeout := Timeout); // FB_MBWriteCoils
WriteCoilsBusy_Modus := LA_955_WriteCoils.bBusy;
WriteCoils_Error_Modus := LA_955_WriteCoils.bError;
WriteCoilsErrID_Modus := LA_955_WriteCoils.nErrId;
Zustand.Betriebsart_Anlage_RM := INT_TO_REAL(LA955_RR_arrData [1]);
_w1 := GETBIT32(inVal32 := LA955_RI_arrData[1], bitNo := 0);
Zustand.Betrieb := _w1;
LA955_WR_arrData[1] := REAL_TO_INT(Zustand.Betriebsartenschalter_Anlage);
_w2 := SETINBYTE(input := 0, bit0 := Steuerung.Anforderung_Lueftung_Seminarraum, bit1 := Steuerung.Anforderung_Lueftung_Halle, bit2 := Steuerung.Entriegelung_Anlage, bit3 := Steuerung.Sollwertauswahl_Anlage, bit4 := Steuerung.Anforderung_Lueftung_Seminarraum_ueber_Nutzungszeit, bit5 := Steuerung.Anforderung_Lueftung_Halle_ueber_Nutzungszeit, bit6 := Steuerung.Anforderung_Lueftung_Seminarraum_ueber_CO2_Grenzwert, bit7 := FALSE);
LA955_WC_arrData[1] := _w2;
Stellwert.Aussenluftklappe_Stellung := INT_TO_REAL(LA955_RR_arrData[2]) / 10;
Zustand.Abluefter_Druck_Istwert := INT_TO_REAL(LA955_RR_arrData[3]) / 10;
Zustand.Abluefter_Drehzahl_Istwert := INT_TO_REAL(LA955_RR_arrData[4]) / 10;
Stellwert.Sollwert_berech_aus_Schiebung := INT_TO_REAL(LA955_RR_arrData[5]) / 10;
Stellwert.Sollwert_aktuell := INT_TO_REAL(LA955_RR_arrData[6]) / 10;
Stellwert.Aussenluftklappe_Stellung := INT_TO_REAL(LA955_RR_arrData[7]) / 10;
Zustand.Ablufttemperatur_Istwert := INT_TO_REAL(LA955_RR_arrData[8]) / 10;
_w3 := GETBIT32(inVal32 := LA955_RI_arrData[1], bitNo := 1);
Zustand.Aussenluftfilterueberwachung := _w3;
_w4 := GETBIT32(inVal32 := LA955_RI_arrData[2], bitNo := 0);
Zustand.Abluftventilator_BM := _w4;
_w5 := GETBIT32(inVal32 := LA955_RI_arrData[3], bitNo := 0);
Zustand.Register_Pumpe_Freigabe := _w5;
_w6 := GETBIT32(inVal32 := LA955_RI_arrData[4], bitNo := 0);
Zustand.Halle_BSK2_offen_RM := _w6;
_w7 := GETBIT32(inVal32 := LA955_RI_arrData[1], bitNo := 2);
Zustand.Abluftfilterueberwachung := _w7;
_w8 := GETBIT32(inVal32 := LA955_RI_arrData[2], bitNo := 1);
Zustand.Abluftventilator_SM := _w8;
_w9 := GETBIT32(inVal32 := LA955_RI_arrData[3], bitNo := 1);
Zustand.Register_Pumpe_Stoerung := _w9;
_w10 := GETBIT32(inVal32 := LA955_RI_arrData[4], bitNo := 1);
Zustand.Seminarraum_BSK1_offen_RM := _w10;
_w11 := GETBIT32(inVal32 := LA955_RI_arrData[1], bitNo := 3);
Zustand.Abluftklappe_oeffnet := _w11;
_w12 := GETBIT32(inVal32 := LA955_RI_arrData[2], bitNo := 2);
Zustand.Abluftventilator_Freigabe := _w12;
_w13 := GETBIT32(inVal32 := LA955_RI_arrData[3], bitNo := 2);
Zustand.Register_Pumpe_BM := _w13;
_w14 := GETBIT32(inVal32 := LA955_RI_arrData[4], bitNo := 2);
Zustand.Seminarraum_BSK2_offen_RM := _w14;
_w15 := GETBIT32(inVal32 := LA955_RI_arrData[1], bitNo := 4);
Zustand.Abluftrauchmelder_SM := _w15;
_w16 := GETBIT32(inVal32 := LA955_RI_arrData[2], bitNo := 3);
Zustand.Change_Overventile_umschalten := _w16;
_w17 := GETBIT32(inVal32 := LA955_RI_arrData[3], bitNo := 3);
Zustand.Brandmeldezentrale_AM := _w17;
_w18 := GETBIT32(inVal32 := LA955_RI_arrData[4], bitNo := 3);
Zustand.Seminarraum_BSK3_offen_RM := _w18;
_w19 := GETBIT32(inVal32 := LA955_RI_arrData[1], bitNo := 5);
Zustand.Abluftrauchmelder_WM := _w19;
_w20 := GETBIT32(inVal32 := LA955_RI_arrData[2], bitNo := 4);
Zustand.Aussenluftklappe_oeffnet := _w20;
_w21 := GETBIT32(inVal32 := LA955_RI_arrData[3], bitNo := 4);
Zustand.Zuluftventilator_BM := _w21;
_w22 := GETBIT32(inVal32 := LA955_RI_arrData[4], bitNo := 4);
Zustand.Seminarraum_BSK_offen_RM := _w22;
_w23 := GETBIT32(inVal32 := LA955_RI_arrData[1], bitNo := 6);
Zustand.Zuluftrauchmelder_SM := _w23;
_w24 := GETBIT32(inVal32 := LA955_RI_arrData[2], bitNo := 5);
Zustand.Option := _w24;
_w25 := GETBIT32(inVal32 := LA955_RI_arrData[3], bitNo := 5);
Zustand.Zuluftventilator_SM := _w25;
_w26 := GETBIT32(inVal32 := LA955_RI_arrData[4], bitNo := 5);
Zustand.Sammelstoerung_Anlage := _w26;
_w27 := GETBIT32(inVal32 := LA955_RI_arrData[1], bitNo := 7);
Zustand.Zuluftrauchmelder_WM := _w27;
_w28 := GETBIT32(inVal32 := LA955_RI_arrData[2], bitNo := 6);
Zustand.Frost_Stoerung := _w28;
_w29 := GETBIT32(inVal32 := LA955_RI_arrData[3], bitNo := 6);
Zustand.Zuluftventilator_Freigabe := _w29;
_w30 := GETBIT32(inVal32 := LA955_RI_arrData[4], bitNo := 6);
Zustand.Sommer_Winter_Umschaltung_Winter_Rueckmeldung := _w30;
_w31 := GETBIT32(inVal32 := LA955_RI_arrData[2], bitNo := 7);
Zustand.Anfahrschaltung_aktiv := _w31;
_w32 := GETBIT32(inVal32 := LA955_RI_arrData[3], bitNo := 7);
Zustand.Halle_BSK1_offen_RM := _w32;
Zustand.Aussenlufttemperatur_Istwert := INT_TO_REAL(LA955_RR_arrData[9]) / 10;
Zustand.Fortlufttemperatur_Istwert := INT_TO_REAL(LA955_RR_arrData[10]) / 10;
Zustand.Zulufttemperatur_Istwert := INT_TO_REAL(LA955_RR_arrData[11]) / 10;
Zustand.Anfahrschaltung_Grenzwert_RL := INT_TO_REAL(LA955_RR_arrData[12]) / 10;
Stellwert.Register_Ventil_Stellung := INT_TO_REAL(LA955_RR_arrData[13]) / 10;
Zustand.Ruecklauftemperatur_Istwert := INT_TO_REAL(LA955_RR_arrData[14]) / 10;
Stellwert.Bypassklappe_Stellung := INT_TO_REAL(LA955_RR_arrData[15]) / 10;
Zustand.Zuluefter_Druck_Istwert := INT_TO_REAL(LA955_RR_arrData[16]) / 10;
Zustand.Zuluefter_Drehzahl_Istwert := INT_TO_REAL(LA955_RR_arrData[17]) / 10;
Zustand.Seminarraum_CO2_Istwert := INT_TO_REAL(LA955_RR_arrData[18]) / 1;
Zustand.Halle_Raumtemperatur_Istwert := INT_TO_REAL(LA955_RR_arrData[19]) / 10;
Zustand.Seminarraum_Raumtemperatur_Istwert := INT_TO_REAL(LA955_RR_arrData[20]) / 10;
Zustand.Halle_Abluft_VSR_Betriebsartenschalter := INT_TO_REAL(LA955_RR_arrData[21]) / 10;
Zustand.Halle_Zuluft_VSR_Betriebsartenschalter := INT_TO_REAL(LA955_RR_arrData[22]) / 10;
Zustand.Seminarraum_Abluft_VSR1_Istwert := INT_TO_REAL(LA955_RR_arrData[23]) / 10;
Zustand.Seminarraum_Zuluft_VSR1_Istwert := INT_TO_REAL(LA955_RR_arrData[24]) / 10;
Zustand.Seminarraum_Abluft_VSR1_Istwert := INT_TO_REAL(LA955_RR_arrData[25]) / 10;
Zustand.Seminarraum_Zuluft_VSR2_Istwert := INT_TO_REAL(LA955_RR_arrData[26]) / 10;
LA955_WR_arrData[2] := REAL_TO_INT(Parameter.Ausschaltverz_Anlage_nach_Taster);
LA955_WR_arrData[18] := REAL_TO_INT(Parameter.Freie_Nachtkuehlung_AT_Grenzwert);
LA955_WR_arrData[34] := REAL_TO_INT(0);
LA955_WR_arrData[3] := REAL_TO_INT(9);
LA955_WR_arrData[19] := REAL_TO_INT(Parameter.Freie_Nachtkuehlung_Diff_AT_zu_RT_Grenzwert);
LA955_WR_arrData[35] := REAL_TO_INT(9);
LA955_WR_arrData[4] := REAL_TO_INT(Parameter.Abluefter_Druck_Sollwert);
LA955_WR_arrData[20] := REAL_TO_INT(Parameter.Freie_Nachtkuehlung_Nacht_Raumsollwert);
LA955_WR_arrData[36] := REAL_TO_INT(0);
LA955_WR_arrData[5] := REAL_TO_INT(9);
LA955_WR_arrData[21] := REAL_TO_INT(Parameter.Zuluefter_Drucksollwert);
LA955_WR_arrData[37] := REAL_TO_INT(9);
LA955_WR_arrData[6] := REAL_TO_INT(0);
LA955_WR_arrData[22] := REAL_TO_INT(9);
LA955_WR_arrData[38] := REAL_TO_INT(0);
LA955_WR_arrData[7] := REAL_TO_INT(9);
LA955_WR_arrData[23] := REAL_TO_INT(9);
LA955_WR_arrData[39] := REAL_TO_INT(Umwelt.Temp_Aussen_WS_Mittelw);
LA955_WR_arrData[8] := REAL_TO_INT(9);
LA955_WR_arrData[24] := REAL_TO_INT(Parameter.Seminarraum_Grenzwert_CO2_Lueftung_Ein);
LA955_WR_arrData[40] := REAL_TO_INT(9);
LA955_WR_arrData[9] := REAL_TO_INT(9);
LA955_WR_arrData[25] := REAL_TO_INT(Parameter.Seminarraum_Grenzwert_CO2_Lueftung_Aus);
LA955_WR_arrData[41] := REAL_TO_INT(18);
LA955_WR_arrData[10] := REAL_TO_INT(0);
LA955_WR_arrData[26] := REAL_TO_INT(Parameter.Seminarraum_CO2_Sollwert_bei_Lueftungsbetrieb);
LA955_WR_arrData[42] := REAL_TO_INT(3);
LA955_WR_arrData[11] := REAL_TO_INT(9);
LA955_WR_arrData[27] := REAL_TO_INT(9);
LA955_WR_arrData[43] := REAL_TO_INT(12);
LA955_WR_arrData[12] := REAL_TO_INT(9);
LA955_WR_arrData[28] := REAL_TO_INT(0);
LA955_WR_arrData[13] := REAL_TO_INT(0);
LA955_WR_arrData[29] := REAL_TO_INT(9);
LA955_WR_arrData[14] := REAL_TO_INT(Parameter.Sollwertschiebung_Anlage_Min_Sollwert);
LA955_WR_arrData[30] := REAL_TO_INT(0);
LA955_WR_arrData[15] := REAL_TO_INT(Parameter.Sollwertschiebung_Anlage_Min_AT_Sollwert);
LA955_WR_arrData[31] := REAL_TO_INT(9);
LA955_WR_arrData[16] := REAL_TO_INT(Parameter.Sollwertschiebung_Anlage_Max_Sollwert);
LA955_WR_arrData[32] := REAL_TO_INT(0);
LA955_WR_arrData[17] := REAL_TO_INT(Parameter.Sollwertschiebung_Anlage_Max_AT_Sollwert);
LA955_WR_arrData[33] := REAL_TO_INT(9);

END_FUNCTION_BLOCK

(* stored: Version 1.1.0.1, ProductVersion 3.1.4024.9
   POU FB_LA: Id {442c14cb-3717-40f4-8c74-0f30a04ba883}, SpecialFunc None *)
